LIN {X 0,Y 566.195,Z 141.956,A -85,B 0,C 180,E1 -2380.2,E2 -2380.2} C_VEL
LIN {X 0,Y 566.194,Z 141.961,A -85,B 0,C 180,E1 -2383.055,E2 -2383.055} C_VEL
LIN {X 0,Y 566.193,Z 141.957,A -85,B 0,C 180,E1 -2386.049,E2 -2386.049} C_VEL
LIN {X 0,Y 566.204,Z 141.954,A -85,B 0,C 180,E1 -2388.865,E2 -2388.865} C_VEL
LIN {X 0,Y 566.171,Z 141.963,A -85,B 0,C 180,E1 -2391.638,E2 -2391.638} C_VEL
LIN {X 0,Y 566.142,Z 141.962,A -85,B 0,C 180,E1 -2394.308,E2 -2394.308} C_VEL
LIN {X 0,Y 566.223,Z 141.954,A -85,B 0,C 180,E1 -2396.9,E2 -2396.9} C_VEL
LIN {X 0,Y 566.19,Z 141.957,A -85,B 0,C 180,E1 -2399.41,E2 -2399.41} C_VEL
LIN {X 0,Y 566.224,Z 141.955,A -85,B 0,C 180,E1 -2401.86,E2 -2401.86} C_VEL
LIN {X 0,Y 566.194,Z 141.955,A -85,B 0,C 180,E1 -2404.252,E2 -2404.252} C_VEL
LIN {X 0,Y 566.159,Z 141.959,A -85,B 0,C 180,E1 -2407.369,E2 -2407.369} C_VEL
LIN {X 0,Y 566.209,Z 141.956,A -85,B 0,C 180,E1 -2409.664,E2 -2409.664} C_VEL
LIN {X 0,Y 566.199,Z 141.955,A -85,B 0,C 180,E1 -2412.67,E2 -2412.67} C_VEL
LIN {X 0,Y 566.213,Z 141.953,A -85,B 0,C 180,E1 -2415.628,E2 -2415.628} C_VEL
LIN {X 0,Y 566.234,Z 141.952,A -85,B 0,C 180,E1 -2418.677,E2 -2418.677} C_VEL
LIN {X 0,Y 566.224,Z 141.954,A -85,B 0,C 180,E1 -2421.435,E2 -2421.435} C_VEL
LIN {X 0,Y 566.261,Z 141.947,A -85,B 0,C 180,E1 -2424.303,E2 -2424.303} C_VEL
LIN {X 0,Y 566.283,Z 141.945,A -85,B 0,C 180,E1 -2427.867,E2 -2427.867} C_VEL
LIN {X 0,Y 566.288,Z 141.949,A -85,B 0,C 180,E1 -2430.001,E2 -2430.001} C_VEL
LIN {X 0,Y 566.258,Z 141.947,A -85,B 0,C 180,E1 -2432.847,E2 -2432.847} C_VEL
LIN {X 0,Y 566.263,Z 141.948,A -85,B 0,C 180,E1 -2435.699,E2 -2435.699} C_VEL
LIN {X 0,Y 566.23,Z 141.956,A -85,B 0,C 180,E1 -2438.567,E2 -2438.567} C_VEL
LIN {X 0,Y 566.243,Z 141.951,A -85,B 0,C 180,E1 -2441.455,E2 -2441.455} C_VEL
LIN {X 0,Y 566.206,Z 141.953,A -85,B 0,C 180,E1 -2444.494,E2 -2444.494} C_VEL
LIN {X 0,Y 566.203,Z 141.956,A -85,B 0,C 180,E1 -2447.332,E2 -2447.332} C_VEL
LIN {X 0,Y 566.212,Z 141.959,A -85,B 0,C 180,E1 -2450.338,E2 -2450.338} C_VEL
LIN {X 0,Y 566.169,Z 141.961,A -85,B 0,C 180,E1 -2453.28,E2 -2453.28} C_VEL
LIN {X 0,Y 566.186,Z 141.957,A -85,B 0,C 180,E1 -2455.751,E2 -2455.751} C_VEL
LIN {X 0,Y 566.157,Z 141.961,A -85,B 0,C 180,E1 -2458.193,E2 -2458.193} C_VEL
LIN {X 0,Y 566.192,Z 141.955,A -85,B 0,C 180,E1 -2461.076,E2 -2461.076} C_VEL
LIN {X 0,Y 566.202,Z 141.96,A -85,B 0,C 180,E1 -2463.732,E2 -2463.732} C_VEL
LIN {X 0,Y 566.183,Z 141.958,A -85,B 0,C 180,E1 -2466.572,E2 -2466.572} C_VEL
LIN {X 0,Y 566.21,Z 141.953,A -85,B 0,C 180,E1 -2469.685,E2 -2469.685} C_VEL
LIN {X 0,Y 566.205,Z 141.954,A -85,B 0,C 180,E1 -2473.055,E2 -2473.055} C_VEL
LIN {X 0,Y 566.198,Z 141.955,A -85,B 0,C 180,E1 -2476.05,E2 -2476.05} C_VEL
LIN {X 0,Y 566.208,Z 141.955,A -85,B 0,C 180,E1 -2479.215,E2 -2479.215} C_VEL
LIN {X 0,Y 566.173,Z 141.958,A -85,B 0,C 180,E1 -2481.636,E2 -2481.636} C_VEL
LIN {X 0,Y 566.153,Z 141.961,A -85,B 0,C 180,E1 -2484.307,E2 -2484.307} C_VEL
LIN {X 0,Y 566.204,Z 141.957,A -85,B 0,C 180,E1 -2486.897,E2 -2486.897} C_VEL
LIN {X 0,Y 566.232,Z 142.057,A -85,B 0,C 180,E1 -2489.617,E2 -2489.617} C_VEL
LIN {X 0,Y 566.413,Z 147.475,A -85,B 0,C 180,E1 -2491.453,E2 -2491.453} C_VEL
LIN {X 0,Y 566.3,Z 155.916,A -85,B 0,C 180,E1 -2494.255,E2 -2494.255} C_VEL
LIN {X 0,Y 566.217,Z 164.488,A -85,B 0,C 180,E1 -2497.043,E2 -2497.043} C_VEL
LIN {X 0,Y 566.168,Z 173.964,A -85,B 0,C 180,E1 -2500.04,E2 -2500.04} C_VEL
LIN {X 0,Y 566.089,Z 183.007,A -85,B 0,C 180,E1 -2502.933,E2 -2502.933} C_VEL
LIN {X 0,Y 566.022,Z 192.721,A -85,B 0,C 180,E1 -2505.988,E2 -2505.988} C_VEL
LIN {X 0,Y 565.964,Z 201.9,A -85,B 0,C 180,E1 -2508.816,E2 -2508.816} C_VEL
LIN {X 0,Y 565.944,Z 211.648,A -85,B 0,C 180,E1 -2511.79,E2 -2511.79} C_VEL
LIN {X 0,Y 565.895,Z 214.384,A -85,B 0,C 180,E1 -2512.619,E2 -2512.619} C_VEL
LIN {X 0,Y 566.251,Z 220.58,A -85,B 0,C 180,E1 -2512.826,E2 -2512.826} C_VEL
LIN {X 0,Y 566.159,Z 229.406,A -85,B 0,C 180,E1 -2513.205,E2 -2513.205} C_VEL
LIN {X 0,Y 566.081,Z 238.598,A -85,B 0,C 180,E1 -2513.764,E2 -2513.764} C_VEL
LIN {X 0,Y 565.989,Z 245.323,A -85,B 0,C 180,E1 -2514.299,E2 -2514.299} C_VEL
LIN {X 0,Y 566.009,Z 252.383,A -85,B 0,C 180,E1 -2515.014,E2 -2515.014} C_VEL
LIN {X 0,Y 565.97,Z 257.771,A -85,B 0,C 180,E1 -2515.727,E2 -2515.727} C_VEL
LIN {X 0,Y 565.969,Z 262.032,A -85,B 0,C 180,E1 -2516.44,E2 -2516.44} C_VEL
LIN {X 0,Y 565.892,Z 265.349,A -85,B 0,C 180,E1 -2517.153,E2 -2517.153} C_VEL
LIN {X 0,Y 565.855,Z 267.84,A -85,B 0,C 180,E1 -2517.865,E2 -2517.865} C_VEL
LIN {X 0,Y 565.847,Z 269.58,A -85,B 0,C 180,E1 -2518.577,E2 -2518.577} C_VEL
LIN {X 0,Y 565.842,Z 270.622,A -85,B 0,C 180,E1 -2519.288,E2 -2519.288} C_VEL
LIN {X 0,Y 565.839,Z 270.996,A -85,B 0,C 180,E1 -2520,E2 -2520} C_VEL
LIN {X 0,Y 565.841,Z 270.711,A -85,B 0,C 180,E1 -2520.712,E2 -2520.712} C_VEL
LIN {X 0,Y 565.848,Z 269.761,A -85,B 0,C 180,E1 -2521.423,E2 -2521.423} C_VEL
LIN {X 0,Y 565.854,Z 268.12,A -85,B 0,C 180,E1 -2522.135,E2 -2522.135} C_VEL
LIN {X 0,Y 565.893,Z 265.732,A -85,B 0,C 180,E1 -2522.848,E2 -2522.848} C_VEL
LIN {X 0,Y 565.991,Z 260.601,A -85,B 0,C 180,E1 -2523.916,E2 -2523.916} C_VEL
LIN {X 0,Y 566.024,Z 254.526,A -85,B 0,C 180,E1 -2524.808,E2 -2524.808} C_VEL
LIN {X 0,Y 565.96,Z 248.211,A -85,B 0,C 180,E1 -2525.523,E2 -2525.523} C_VEL
LIN {X 0,Y 566.069,Z 241.059,A -85,B 0,C 180,E1 -2526.147,E2 -2526.147} C_VEL
LIN {X 0,Y 566.09,Z 233.058,A -85,B 0,C 180,E1 -2526.683,E2 -2526.683} C_VEL
LIN {X 0,Y 566.211,Z 224.178,A -85,B 0,C 180,E1 -2527.13,E2 -2527.13} C_VEL
LIN {X 0,Y 566.062,Z 216.549,A -85,B 0,C 180,E1 -2527.401,E2 -2527.401} C_VEL
LIN {X 0,Y 565.899,Z 214.311,A -85,B 0,C 180,E1 -2527.493,E2 -2527.493} C_VEL
LIN {X 0,Y 565.944,Z 204.843,A -85,B 0,C 180,E1 -2530.374,E2 -2530.374} C_VEL
LIN {X 0,Y 566.004,Z 195.375,A -85,B 0,C 180,E1 -2533.28,E2 -2533.28} C_VEL
LIN {X 0,Y 566.052,Z 187.164,A -85,B 0,C 180,E1 -2535.852,E2 -2535.852} C_VEL
LIN {X 0,Y 566.16,Z 177.828,A -85,B 0,C 180,E1 -2538.829,E2 -2538.829} C_VEL
LIN {X 0,Y 566.197,Z 168.251,A -85,B 0,C 180,E1 -2541.863,E2 -2541.863} C_VEL
LIN {X 0,Y 566.261,Z 158.561,A -85,B 0,C 180,E1 -2544.96,E2 -2544.96} C_VEL
LIN {X 0,Y 566.335,Z 149.951,A -85,B 0,C 180,E1 -2547.734,E2 -2547.734} C_VEL
LIN {X 0,Y 566.402,Z 143.716,A -85,B 0,C 180,E1 -2549.757,E2 -2549.757} C_VEL
LIN {X 0,Y 566.261,Z 141.954,A -85,B 0,C 180,E1 -2550.382,E2 -2550.382} C_VEL
LIN {X 0,Y 566.208,Z 141.958,A -85,B 0,C 180,E1 -2553.103,E2 -2553.103} C_VEL
LIN {X 0,Y 566.168,Z 141.964,A -85,B 0,C 180,E1 -2555.692,E2 -2555.692} C_VEL
LIN {X 0,Y 566.215,Z 141.957,A -85,B 0,C 180,E1 -2558.558,E2 -2558.558} C_VEL
LIN {X 0,Y 566.178,Z 141.962,A -85,B 0,C 180,E1 -2561.14,E2 -2561.14} C_VEL
LIN {X 0,Y 566.198,Z 141.959,A -85,B 0,C 180,E1 -2564.036,E2 -2564.036} C_VEL
LIN {X 0,Y 566.208,Z 141.959,A -85,B 0,C 180,E1 -2567.082,E2 -2567.082} C_VEL
LIN {X 0,Y 566.219,Z 141.958,A -85,B 0,C 180,E1 -2570.314,E2 -2570.314} C_VEL
LIN {X 0,Y 566.205,Z 141.96,A -85,B 0,C 180,E1 -2573.43,E2 -2573.43} C_VEL
LIN {X 0,Y 566.204,Z 141.959,A -85,B 0,C 180,E1 -2576.268,E2 -2576.268} C_VEL
LIN {X 0,Y 566.197,Z 141.963,A -85,B 0,C 180,E1 -2578.923,E2 -2578.923} C_VEL
LIN {X 0,Y 566.218,Z 141.96,A -85,B 0,C 180,E1 -2581.857,E2 -2581.857} C_VEL
LIN {X 0,Y 566.268,Z 142.067,A -85,B 0,C 180,E1 -2582.262,E2 -2582.262} C_VEL
LIN {X 0,Y 567.185,Z 147.623,A -85,B 0,C 180,E1 -2583.507,E2 -2583.507} C_VEL
LIN {X 0,Y 566.963,Z 159.309,A -85,B 0,C 180,E1 -2585.853,E2 -2585.853} C_VEL
LIN {X 0,Y 566.676,Z 173.884,A -85,B 0,C 180,E1 -2588.687,E2 -2588.687} C_VEL
LIN {X 0,Y 566.475,Z 189.392,A -85,B 0,C 180,E1 -2591.556,E2 -2591.556} C_VEL
LIN {X 0,Y 566.325,Z 204.592,A -85,B 0,C 180,E1 -2594.34,E2 -2594.34} C_VEL
LIN {X 0,Y 566.205,Z 219.792,A -85,B 0,C 180,E1 -2597.089,E2 -2597.089} C_VEL
LIN {X 0,Y 566.177,Z 221.014,A -85,B 0,C 180,E1 -2597.293,E2 -2597.293} C_VEL
LIN {X 0,Y 566.981,Z 226.896,A -85,B 0,C 180,E1 -2597.403,E2 -2597.403} C_VEL
LIN {X 0,Y 566.85,Z 239.423,A -85,B 0,C 180,E1 -2597.695,E2 -2597.695} C_VEL
LIN {X 0,Y 566.733,Z 252.352,A -85,B 0,C 180,E1 -2598.147,E2 -2598.147} C_VEL
LIN {X 0,Y 566.594,Z 264.395,A -85,B 0,C 180,E1 -2598.721,E2 -2598.721} C_VEL
LIN {X 0,Y 566.457,Z 276.184,A -85,B 0,C 180,E1 -2599.454,E2 -2599.454} C_VEL
LIN {X 0,Y 566.327,Z 286.591,A -85,B 0,C 180,E1 -2600.264,E2 -2600.264} C_VEL
LIN {X 0,Y 566.207,Z 295.103,A -85,B 0,C 180,E1 -2601.073,E2 -2601.073} C_VEL
LIN {X 0,Y 566.113,Z 302.952,A -85,B 0,C 180,E1 -2601.971,E2 -2601.971} C_VEL
LIN {X 0,Y 566.005,Z 310.616,A -85,B 0,C 180,E1 -2603.046,E2 -2603.046} C_VEL
LIN {X 0,Y 566.004,Z 317.674,A -85,B 0,C 180,E1 -2604.298,E2 -2604.298} C_VEL
LIN {X 0,Y 565.933,Z 322.368,A -85,B 0,C 180,E1 -2605.369,E2 -2605.369} C_VEL
LIN {X 0,Y 565.927,Z 325.955,A -85,B 0,C 180,E1 -2606.439,E2 -2606.439} C_VEL
LIN {X 0,Y 565.878,Z 327.805,A -85,B 0,C 180,E1 -2607.151,E2 -2607.151} C_VEL
LIN {X 0,Y 565.846,Z 330.183,A -85,B 0,C 180,E1 -2608.575,E2 -2608.575} C_VEL
LIN {X 0,Y 565.839,Z 331,A -85,B 0,C 180,E1 -2609.999,E2 -2609.999} C_VEL
LIN {X 0,Y 565.846,Z 330.187,A -85,B 0,C 180,E1 -2611.422,E2 -2611.422} C_VEL
LIN {X 0,Y 565.877,Z 327.813,A -85,B 0,C 180,E1 -2612.846,E2 -2612.846} C_VEL
LIN {X 0,Y 565.926,Z 324.9,A -85,B 0,C 180,E1 -2613.915,E2 -2613.915} C_VEL
LIN {X 0,Y 565.877,Z 320.954,A -85,B 0,C 180,E1 -2614.986,E2 -2614.986} C_VEL
LIN {X 0,Y 566.007,Z 315.874,A -85,B 0,C 180,E1 -2616.057,E2 -2616.057} C_VEL
LIN {X 0,Y 566.039,Z 309.476,A -85,B 0,C 180,E1 -2617.131,E2 -2617.131} C_VEL
LIN {X 0,Y 566.133,Z 301.488,A -85,B 0,C 180,E1 -2618.206,E2 -2618.206} C_VEL
LIN {X 0,Y 566.228,Z 293.347,A -85,B 0,C 180,E1 -2619.104,E2 -2619.104} C_VEL
LIN {X 0,Y 566.34,Z 283.415,A -85,B 0,C 180,E1 -2620.004,E2 -2620.004} C_VEL
LIN {X 0,Y 566.519,Z 272.33,A -85,B 0,C 180,E1 -2620.805,E2 -2620.805} C_VEL
LIN {X 0,Y 566.61,Z 261.199,A -85,B 0,C 180,E1 -2621.445,E2 -2621.445} C_VEL
LIN {X 0,Y 566.738,Z 249.013,A -85,B 0,C 180,E1 -2621.987,E2 -2621.987} C_VEL
LIN {X 0,Y 566.857,Z 236.227,A -85,B 0,C 180,E1 -2622.393,E2 -2622.393} C_VEL
LIN {X 0,Y 566.84,Z 225.151,A -85,B 0,C 180,E1 -2622.629,E2 -2622.629} C_VEL
LIN {X 0,Y 566.184,Z 220.818,A -85,B 0,C 180,E1 -2622.727,E2 -2622.727} C_VEL
LIN {X 0,Y 566.298,Z 205.618,A -85,B 0,C 180,E1 -2625.474,E2 -2625.474} C_VEL
LIN {X 0,Y 566.449,Z 190.418,A -85,B 0,C 180,E1 -2628.256,E2 -2628.256} C_VEL
LIN {X 0,Y 566.615,Z 177.294,A -85,B 0,C 180,E1 -2630.7,E2 -2630.7} C_VEL
LIN {X 0,Y 566.822,Z 164.181,A -85,B 0,C 180,E1 -2633.181,E2 -2633.181} C_VEL
LIN {X 0,Y 567.057,Z 150.067,A -85,B 0,C 180,E1 -2635.904,E2 -2635.904} C_VEL
LIN {X 0,Y 566.769,Z 144.561,A -85,B 0,C 180,E1 -2637.002,E2 -2637.002} C_VEL
LIN {X 0,Y 566.238,Z 141.954,A -85,B 0,C 180,E1 -2637.587,E2 -2637.587} C_VEL
LIN {X 0,Y 566.163,Z 141.965,A -85,B 0,C 180,E1 -2640.592,E2 -2640.592} C_VEL
LIN {X 0,Y 566.223,Z 141.952,A -85,B 0,C 180,E1 -2643.1,E2 -2643.1} C_VEL
LIN {X 0,Y 566.208,Z 141.96,A -85,B 0,C 180,E1 -2645.687,E2 -2645.687} C_VEL
LIN {X 0,Y 566.204,Z 141.955,A -85,B 0,C 180,E1 -2648.557,E2 -2648.557} C_VEL
LIN {X 0,Y 566.157,Z 141.962,A -85,B 0,C 180,E1 -2651.139,E2 -2651.139} C_VEL
LIN {X 0,Y 566.184,Z 141.961,A -85,B 0,C 180,E1 -2654.035,E2 -2654.035} C_VEL
LIN {X 0,Y 566.196,Z 141.957,A -85,B 0,C 180,E1 -2657.081,E2 -2657.081} C_VEL
LIN {X 0,Y 566.217,Z 141.953,A -85,B 0,C 180,E1 -2659.802,E2 -2659.802} C_VEL
LIN {X 0,Y 566.181,Z 141.963,A -85,B 0,C 180,E1 -2662.599,E2 -2662.599} C_VEL
LIN {X 0,Y 566.195,Z 141.96,A -85,B 0,C 180,E1 -2666.043,E2 -2666.043} C_VEL
LIN {X 0,Y 566.193,Z 141.955,A -85,B 0,C 180,E1 -2668.578,E2 -2668.578} C_VEL
LIN {X 0,Y 566.186,Z 141.962,A -85,B 0,C 180,E1 -2671.046,E2 -2671.046} C_VEL
LIN {X 0,Y 566.235,Z 141.95,A -85,B 0,C 180,E1 -2673.46,E2 -2673.46} C_VEL
LIN {X 0,Y 566.183,Z 141.961,A -85,B 0,C 180,E1 -2675.818,E2 -2675.818} C_VEL
LIN {X 0,Y 566.194,Z 141.956,A -85,B 0,C 180,E1 -2678.902,E2 -2678.902} C_VEL
LIN {X 0,Y 566.201,Z 141.959,A -85,B 0,C 180,E1 -2681.172,E2 -2681.172} C_VEL
LIN {X 0,Y 566.211,Z 141.953,A -85,B 0,C 180,E1 -2683.412,E2 -2683.412} C_VEL
LIN {X 0,Y 566.191,Z 141.958,A -85,B 0,C 180,E1 -2686.359,E2 -2686.359} C_VEL
LIN {X 0,Y 566.218,Z 141.952,A -85,B 0,C 180,E1 -2688.675,E2 -2688.675} C_VEL
LIN {X 0,Y 566.205,Z 141.956,A -85,B 0,C 180,E1 -2691.434,E2 -2691.434} C_VEL
LIN {X 0,Y 566.249,Z 141.953,A -85,B 0,C 180,E1 -2694.302,E2 -2694.302} C_VEL
LIN {X 0,Y 566.27,Z 141.951,A -85,B 0,C 180,E1 -2697.866,E2 -2697.866} C_VEL
LIN {X 0,Y 566.286,Z 141.945,A -85,B 0,C 180,E1 -2700.711,E2 -2700.711} C_VEL
LIN {X 0,Y 566.16,Z 141.959,A -85,B 0,C 180,E1 -2703.558,E2 -2703.558} C_VEL
LIN {X 0,Y 566.243,Z 141.95,A -85,B 0,C 180,E1 -2705.698,E2 -2705.698} C_VEL
LIN {X 0,Y 566.239,Z 141.95,A -85,B 0,C 180,E1 -2708.566,E2 -2708.566} C_VEL
LIN {X 0,Y 566.236,Z 141.954,A -85,B 0,C 180,E1 -2711.454,E2 -2711.454} C_VEL
LIN {X 0,Y 566.213,Z 141.958,A -85,B 0,C 180,E1 -2714.505,E2 -2714.505} C_VEL
LIN {X 0,Y 566.19,Z 141.956,A -85,B 0,C 180,E1 -2717.332,E2 -2717.332} C_VEL
LIN {X 0,Y 566.207,Z 141.954,A -85,B 0,C 180,E1 -2720.337,E2 -2720.337} C_VEL
LIN {X 0,Y 566.217,Z 141.954,A -85,B 0,C 180,E1 -2723.403,E2 -2723.403} C_VEL
LIN {X 0,Y 566.192,Z 141.956,A -85,B 0,C 180,E1 -2725.75,E2 -2725.75} C_VEL
LIN {X 0,Y 566.149,Z 141.96,A -85,B 0,C 180,E1 -2727.502,E2 -2727.502} C_VEL
LIN {X 0,Y 565.482,Z 142.049,A -85,B 0,C 180,E1 -2728.096,E2 -2728.096} C_VEL
LIN {X 0,Y 562.634,Z 142.399,A -85,B 0,C 180,E1 -2729.06,E2 -2729.06} C_VEL
LIN {X 0,Y 560.235,Z 142.702,A -85,B 0,C 180,E1 -2729.836,E2 -2729.836} C_VEL
LIN {X 0,Y 559.214,Z 142.825,A -85,B 0,C 180,E1 -2730.435,E2 -2730.435} C_VEL
LIN {X 0,Y 559.136,Z 142.834,A -85,B 0,C 180,E1 -2730.638,E2 -2730.638} C_VEL
LIN {X 0,Y 559.166,Z 142.832,A -85,B 0,C 180,E1 -2733.575,E2 -2733.575} C_VEL
LIN {X 0,Y 559.158,Z 142.837,A -85,B 0,C 180,E1 -2736.45,E2 -2736.45} C_VEL
LIN {X 0,Y 559.161,Z 142.831,A -85,B 0,C 180,E1 -2738.935,E2 -2738.935} C_VEL
LIN {X 0,Y 559.151,Z 142.835,A -85,B 0,C 180,E1 -2741.771,E2 -2741.771} C_VEL
LIN {X 0,Y 559.145,Z 142.834,A -85,B 0,C 180,E1 -2744.241,E2 -2744.241} C_VEL
LIN {X 0,Y 559.155,Z 142.832,A -85,B 0,C 180,E1 -2747.258,E2 -2747.258} C_VEL
LIN {X 0,Y 559.171,Z 142.833,A -85,B 0,C 180,E1 -2750.136,E2 -2750.136} C_VEL
LIN {X 0,Y 559.122,Z 142.839,A -85,B 0,C 180,E1 -2752.892,E2 -2752.892} C_VEL
LIN {X 0,Y 559.16,Z 142.832,A -85,B 0,C 180,E1 -2756.052,E2 -2756.052} C_VEL
LIN {X 0,Y 559.162,Z 142.831,A -85,B 0,C 180,E1 -2758.983,E2 -2758.983} C_VEL
LIN {X 0,Y 559.164,Z 142.836,A -85,B 0,C 180,E1 -2761.62,E2 -2761.62} C_VEL
LIN {X 0,Y 559.167,Z 142.83,A -85,B 0,C 180,E1 -2763.904,E2 -2763.904} C_VEL
LIN {X 0,Y 559.107,Z 142.839,A -85,B 0,C 180,E1 -2767.068,E2 -2767.068} C_VEL
LIN {X 0,Y 559.176,Z 142.83,A -85,B 0,C 180,E1 -2769.397,E2 -2769.397} C_VEL
LIN {X 0,Y 559.146,Z 142.839,A -85,B 0,C 180,E1 -2771.687,E2 -2771.687} C_VEL
LIN {X 0,Y 559.163,Z 142.832,A -85,B 0,C 180,E1 -2773.949,E2 -2773.949} C_VEL
LIN {X 0,Y 559.149,Z 142.834,A -85,B 0,C 180,E1 -2776.185,E2 -2776.185} C_VEL
LIN {X 0,Y 559.19,Z 142.827,A -85,B 0,C 180,E1 -2779.135,E2 -2779.135} C_VEL
LIN {X 0,Y 559.2,Z 142.829,A -85,B 0,C 180,E1 -2782.055,E2 -2782.055} C_VEL
LIN {X 0,Y 559.252,Z 142.825,A -85,B 0,C 180,E1 -2784.955,E2 -2784.955} C_VEL
LIN {X 0,Y 559.254,Z 142.82,A -85,B 0,C 180,E1 -2787.841,E2 -2787.841} C_VEL
LIN {X 0,Y 559.256,Z 142.824,A -85,B 0,C 180,E1 -2790.001,E2 -2790.001} C_VEL
LIN {X 0,Y 559.226,Z 142.823,A -85,B 0,C 180,E1 -2792.883,E2 -2792.883} C_VEL
LIN {X 0,Y 559.232,Z 142.823,A -85,B 0,C 180,E1 -2795.771,E2 -2795.771} C_VEL
LIN {X 0,Y 559.188,Z 142.833,A -85,B 0,C 180,E1 -2798.675,E2 -2798.675} C_VEL
LIN {X 0,Y 559.2,Z 142.83,A -85,B 0,C 180,E1 -2801.602,E2 -2801.602} C_VEL
LIN {X 0,Y 559.156,Z 142.832,A -85,B 0,C 180,E1 -2804.577,E2 -2804.577} C_VEL
LIN {X 0,Y 559.146,Z 142.833,A -85,B 0,C 180,E1 -2807.558,E2 -2807.558} C_VEL
LIN {X 0,Y 559.171,Z 142.832,A -85,B 0,C 180,E1 -2809.838,E2 -2809.838} C_VEL
LIN {X 0,Y 559.137,Z 142.838,A -85,B 0,C 180,E1 -2812.154,E2 -2812.154} C_VEL
LIN {X 0,Y 559.142,Z 142.839,A -85,B 0,C 180,E1 -2815.178,E2 -2815.178} C_VEL
LIN {X 0,Y 559.119,Z 142.836,A -85,B 0,C 180,E1 -2817.716,E2 -2817.716} C_VEL
LIN {X 0,Y 559.143,Z 142.838,A -85,B 0,C 180,E1 -2820.184,E2 -2820.184} C_VEL
LIN {X 0,Y 559.157,Z 142.832,A -85,B 0,C 180,E1 -2822.716,E2 -2822.716} C_VEL
LIN {X 0,Y 559.128,Z 142.842,A -85,B 0,C 180,E1 -2825.325,E2 -2825.325} C_VEL
LIN {X 0,Y 559.11,Z 142.837,A -85,B 0,C 180,E1 -2828.02,E2 -2828.02} C_VEL
LIN {X 0,Y 559.159,Z 142.832,A -85,B 0,C 180,E1 -2829.941,E2 -2829.941} C_VEL
LIN {X 0,Y 559.161,Z 142.832,A -85,B 0,C 180,E1 -2832.744,E2 -2832.744} C_VEL
LIN {X 0,Y 559.152,Z 142.835,A -85,B 0,C 180,E1 -2835.762,E2 -2835.762} C_VEL
LIN {X 0,Y 559.166,Z 142.831,A -85,B 0,C 180,E1 -2838.23,E2 -2838.23} C_VEL
LIN {X 0,Y 559.169,Z 142.829,A -85,B 0,C 180,E1 -2841.193,E2 -2841.193} C_VEL
LIN {X 0,Y 559.123,Z 142.842,A -85,B 0,C 180,E1 -2843.788,E2 -2843.788} C_VEL
LIN {X 0,Y 559.151,Z 142.833,A -85,B 0,C 180,E1 -2846.424,E2 -2846.424} C_VEL
LIN {X 0,Y 559.213,Z 142.917,A -85,B 0,C 180,E1 -2849.508,E2 -2849.508} C_VEL
LIN {X 0,Y 559.399,Z 147.468,A -85,B 0,C 180,E1 -2851.073,E2 -2851.073} C_VEL
LIN {X 0,Y 559.291,Z 155.893,A -85,B 0,C 180,E1 -2853.908,E2 -2853.908} C_VEL
LIN {X 0,Y 559.165,Z 163.968,A -85,B 0,C 180,E1 -2856.567,E2 -2856.567} C_VEL
LIN {X 0,Y 559.132,Z 172.758,A -85,B 0,C 180,E1 -2859.394,E2 -2859.394} C_VEL
LIN {X 0,Y 559.041,Z 181.068,A -85,B 0,C 180,E1 -2862.061,E2 -2862.061} C_VEL
LIN {X 0,Y 558.988,Z 189.275,A -85,B 0,C 180,E1 -2864.691,E2 -2864.691} C_VEL
LIN {X 0,Y 558.935,Z 197.495,A -85,B 0,C 180,E1 -2867.288,E2 -2867.288} C_VEL
LIN {X 0,Y 558.864,Z 206.917,A -85,B 0,C 180,E1 -2870.226,E2 -2870.226} C_VEL
LIN {X 0,Y 558.832,Z 214.386,A -85,B 0,C 180,E1 -2872.526,E2 -2872.526} C_VEL
LIN {X 0,Y 559.208,Z 221.803,A -85,B 0,C 180,E1 -2872.78,E2 -2872.78} C_VEL
LIN {X 0,Y 559.111,Z 230.589,A -85,B 0,C 180,E1 -2873.178,E2 -2873.178} C_VEL
LIN {X 0,Y 559.039,Z 238.604,A -85,B 0,C 180,E1 -2873.685,E2 -2873.685} C_VEL
LIN {X 0,Y 558.935,Z 245.327,A -85,B 0,C 180,E1 -2874.227,E2 -2874.227} C_VEL
LIN {X 0,Y 558.929,Z 252.388,A -85,B 0,C 180,E1 -2874.95,E2 -2874.95} C_VEL
LIN {X 0,Y 558.907,Z 257.774,A -85,B 0,C 180,E1 -2875.673,E2 -2875.673} C_VEL
LIN {X 0,Y 558.882,Z 262.035,A -85,B 0,C 180,E1 -2876.395,E2 -2876.395} C_VEL
LIN {X 0,Y 558.816,Z 265.352,A -85,B 0,C 180,E1 -2877.116,E2 -2877.116} C_VEL
LIN {X 0,Y 558.763,Z 267.843,A -85,B 0,C 180,E1 -2877.838,E2 -2877.838} C_VEL
LIN {X 0,Y 558.747,Z 269.582,A -85,B 0,C 180,E1 -2878.559,E2 -2878.559} C_VEL
LIN {X 0,Y 558.742,Z 270.623,A -85,B 0,C 180,E1 -2879.279,E2 -2879.279} C_VEL
LIN {X 0,Y 558.74,Z 270.996,A -85,B 0,C 180,E1 -2880,E2 -2880} C_VEL
LIN {X 0,Y 558.741,Z 270.71,A -85,B 0,C 180,E1 -2880.721,E2 -2880.721} C_VEL
LIN {X 0,Y 558.748,Z 269.759,A -85,B 0,C 180,E1 -2881.442,E2 -2881.442} C_VEL
LIN {X 0,Y 558.763,Z 268.118,A -85,B 0,C 180,E1 -2882.163,E2 -2882.163} C_VEL
LIN {X 0,Y 558.816,Z 265.73,A -85,B 0,C 180,E1 -2882.884,E2 -2882.884} C_VEL
LIN {X 0,Y 558.89,Z 260.598,A -85,B 0,C 180,E1 -2883.966,E2 -2883.966} C_VEL
LIN {X 0,Y 558.952,Z 254.521,A -85,B 0,C 180,E1 -2884.869,E2 -2884.869} C_VEL
LIN {X 0,Y 558.896,Z 248.204,A -85,B 0,C 180,E1 -2885.593,E2 -2885.593} C_VEL
LIN {X 0,Y 559.025,Z 241.053,A -85,B 0,C 180,E1 -2886.225,E2 -2886.225} C_VEL
LIN {X 0,Y 559.037,Z 232.936,A -85,B 0,C 180,E1 -2886.775,E2 -2886.775} C_VEL
LIN {X 0,Y 559.176,Z 224.165,A -85,B 0,C 180,E1 -2887.22,E2 -2887.22} C_VEL
LIN {X 0,Y 558.931,Z 215.697,A -85,B 0,C 180,E1 -2887.519,E2 -2887.519} C_VEL
LIN {X 0,Y 558.803,Z 214.309,A -85,B 0,C 180,E1 -2887.589,E2 -2887.589} C_VEL
LIN {X 0,Y 558.863,Z 204.841,A -85,B 0,C 180,E1 -2890.506,E2 -2890.506} C_VEL
LIN {X 0,Y 558.94,Z 195.462,A -85,B 0,C 180,E1 -2893.451,E2 -2893.451} C_VEL
LIN {X 0,Y 559.03,Z 186.106,A -85,B 0,C 180,E1 -2896.431,E2 -2896.431} C_VEL
LIN {X 0,Y 559.108,Z 177.94,A -85,B 0,C 180,E1 -2899.076,E2 -2899.076} C_VEL
LIN {X 0,Y 559.145,Z 170.146,A -85,B 0,C 180,E1 -2901.545,E2 -2901.545} C_VEL
LIN {X 0,Y 559.247,Z 160.994,A -85,B 0,C 180,E1 -2904.501,E2 -2904.501} C_VEL
LIN {X 0,Y 559.327,Z 152.415,A -85,B 0,C 180,E1 -2907.299,E2 -2907.299} C_VEL
LIN {X 0,Y 559.389,Z 144.546,A -85,B 0,C 180,E1 -2909.899,E2 -2909.899} C_VEL
LIN {X 0,Y 559.191,Z 142.834,A -85,B 0,C 180,E1 -2910.494,E2 -2910.494} C_VEL
LIN {X 0,Y 559.153,Z 142.838,A -85,B 0,C 180,E1 -2913.576,E2 -2913.576} C_VEL
LIN {X 0,Y 559.152,Z 142.837,A -85,B 0,C 180,E1 -2916.445,E2 -2916.445} C_VEL
LIN {X 0,Y 559.179,Z 142.834,A -85,B 0,C 180,E1 -2918.934,E2 -2918.934} C_VEL
LIN {X 0,Y 559.168,Z 142.835,A -85,B 0,C 180,E1 -2921.77,E2 -2921.77} C_VEL
LIN {X 0,Y 559.141,Z 142.84,A -85,B 0,C 180,E1 -2924.739,E2 -2924.739} C_VEL
LIN {X 0,Y 559.164,Z 142.835,A -85,B 0,C 180,E1 -2927.256,E2 -2927.256} C_VEL
LIN {X 0,Y 559.184,Z 142.835,A -85,B 0,C 180,E1 -2930.134,E2 -2930.134} C_VEL
LIN {X 0,Y 559.146,Z 142.837,A -85,B 0,C 180,E1 -2932.891,E2 -2932.891} C_VEL
LIN {X 0,Y 559.163,Z 142.836,A -85,B 0,C 180,E1 -2936.052,E2 -2936.052} C_VEL
LIN {X 0,Y 559.161,Z 142.84,A -85,B 0,C 180,E1 -2938.98,E2 -2938.98} C_VEL
LIN {X 0,Y 559.209,Z 142.911,A -85,B 0,C 180,E1 -2941.987,E2 -2941.987} C_VEL
LIN {X 0,Y 560.154,Z 147.894,A -85,B 0,C 180,E1 -2943.148,E2 -2943.148} C_VEL
LIN {X 0,Y 560.181,Z 154.731,A -85,B 0,C 180,E1 -2944.597,E2 -2944.597} C_VEL
LIN {X 0,Y 559.838,Z 167.218,A -85,B 0,C 180,E1 -2947.097,E2 -2947.097} C_VEL
LIN {X 0,Y 559.603,Z 182.102,A -85,B 0,C 180,E1 -2949.986,E2 -2949.986} C_VEL
LIN {X 0,Y 559.403,Z 196.824,A -85,B 0,C 180,E1 -2952.712,E2 -2952.712} C_VEL
LIN {X 0,Y 559.17,Z 212.202,A -85,B 0,C 180,E1 -2955.535,E2 -2955.535} C_VEL
LIN {X 0,Y 559.169,Z 221.014,A -85,B 0,C 180,E1 -2957.131,E2 -2957.131} C_VEL
LIN {X 0,Y 560.049,Z 228.038,A -85,B 0,C 180,E1 -2957.267,E2 -2957.267} C_VEL
LIN {X 0,Y 559.919,Z 240.946,A -85,B 0,C 180,E1 -2957.586,E2 -2957.586} C_VEL
LIN {X 0,Y 559.766,Z 253.473,A -85,B 0,C 180,E1 -2958.043,E2 -2958.043} C_VEL
LIN {X 0,Y 559.628,Z 265.407,A -85,B 0,C 180,E1 -2958.637,E2 -2958.637} C_VEL
LIN {X 0,Y 559.427,Z 277.472,A -85,B 0,C 180,E1 -2959.412,E2 -2959.412} C_VEL
LIN {X 0,Y 559.298,Z 287.635,A -85,B 0,C 180,E1 -2960.232,E2 -2960.232} C_VEL
LIN {X 0,Y 559.133,Z 296.777,A -85,B 0,C 180,E1 -2961.142,E2 -2961.142} C_VEL
LIN {X 0,Y 559.01,Z 305.681,A -85,B 0,C 180,E1 -2962.232,E2 -2962.232} C_VEL
LIN {X 0,Y 558.926,Z 311.733,A -85,B 0,C 180,E1 -2963.139,E2 -2963.139} C_VEL
LIN {X 0,Y 558.936,Z 317.674,A -85,B 0,C 180,E1 -2964.226,E2 -2964.226} C_VEL
LIN {X 0,Y 558.827,Z 322.368,A -85,B 0,C 180,E1 -2965.31,E2 -2965.31} C_VEL
LIN {X 0,Y 558.836,Z 325.955,A -85,B 0,C 180,E1 -2966.394,E2 -2966.394} C_VEL
LIN {X 0,Y 558.799,Z 327.805,A -85,B 0,C 180,E1 -2967.115,E2 -2967.115} C_VEL
LIN {X 0,Y 558.745,Z 330.182,A -85,B 0,C 180,E1 -2968.557,E2 -2968.557} C_VEL
LIN {X 0,Y 558.74,Z 331,A -85,B 0,C 180,E1 -2969.999,E2 -2969.999} C_VEL
LIN {X 0,Y 558.745,Z 330.186,A -85,B 0,C 180,E1 -2971.44,E2 -2971.44} C_VEL
LIN {X 0,Y 558.799,Z 327.813,A -85,B 0,C 180,E1 -2972.882,E2 -2972.882} C_VEL
LIN {X 0,Y 558.844,Z 324.899,A -85,B 0,C 180,E1 -2973.965,E2 -2973.965} C_VEL
LIN {X 0,Y 558.798,Z 320.954,A -85,B 0,C 180,E1 -2975.05,E2 -2975.05} C_VEL
LIN {X 0,Y 558.922,Z 315.874,A -85,B 0,C 180,E1 -2976.134,E2 -2976.134} C_VEL
LIN {X 0,Y 558.976,Z 309.475,A -85,B 0,C 180,E1 -2977.222,E2 -2977.222} C_VEL
LIN {X 0,Y 559.098,Z 301.488,A -85,B 0,C 180,E1 -2978.31,E2 -2978.31} C_VEL
LIN {X 0,Y 559.194,Z 293.346,A -85,B 0,C 180,E1 -2979.22,E2 -2979.22} C_VEL
LIN {X 0,Y 559.349,Z 283.414,A -85,B 0,C 180,E1 -2980.13,E2 -2980.13} C_VEL
LIN {X 0,Y 559.541,Z 272.427,A -85,B 0,C 180,E1 -2980.935,E2 -2980.935} C_VEL
LIN {X 0,Y 559.669,Z 260.484,A -85,B 0,C 180,E1 -2981.626,E2 -2981.626} C_VEL
LIN {X 0,Y 559.826,Z 247.804,A -85,B 0,C 180,E1 -2982.183,E2 -2982.183} C_VEL
LIN {X 0,Y 559.969,Z 234.397,A -85,B 0,C 180,E1 -2982.594,E2 -2982.594} C_VEL
LIN {X 0,Y 559.846,Z 225.694,A -85,B 0,C 180,E1 -2982.781,E2 -2982.781} C_VEL
LIN {X 0,Y 559.151,Z 220.818,A -85,B 0,C 180,E1 -2982.89,E2 -2982.89} C_VEL
LIN {X 0,Y 559.292,Z 205.618,A -85,B 0,C 180,E1 -2985.673,E2 -2985.673} C_VEL
LIN {X 0,Y 559.453,Z 190.304,A -85,B 0,C 180,E1 -2988.492,E2 -2988.492} C_VEL
LIN {X 0,Y 559.671,Z 177.281,A -85,B 0,C 180,E1 -2990.969,E2 -2990.969} C_VEL
LIN {X 0,Y 559.892,Z 165.414,A -85,B 0,C 180,E1 -2993.256,E2 -2993.256} C_VEL
LIN {X 0,Y 560.127,Z 153.074,A -85,B 0,C 180,E1 -2995.662,E2 -2995.662} C_VEL
LIN {X 0,Y 559.919,Z 146.518,A -85,B 0,C 180,E1 -2996.978,E2 -2996.978} C_VEL
LIN {X 0,Y 559.172,Z 142.835,A -85,B 0,C 180,E1 -2997.811,E2 -2997.811} C_VEL
LIN {X 0,Y 559.145,Z 142.837,A -85,B 0,C 180,E1 -3001.018,E2 -3001.018} C_VEL
LIN {X 0,Y 559.163,Z 142.836,A -85,B 0,C 180,E1 -3003.948,E2 -3003.948} C_VEL
LIN {X 0,Y 559.164,Z 142.831,A -85,B 0,C 180,E1 -3006.447,E2 -3006.447} C_VEL
LIN {X 0,Y 559.167,Z 142.835,A -85,B 0,C 180,E1 -3008.933,E2 -3008.933} C_VEL
LIN {X 0,Y 559.145,Z 142.833,A -85,B 0,C 180,E1 -3011.77,E2 -3011.77} C_VEL
LIN {X 0,Y 559.129,Z 142.836,A -85,B 0,C 180,E1 -3014.738,E2 -3014.738} C_VEL
LIN {X 0,Y 559.155,Z 142.836,A -85,B 0,C 180,E1 -3017.256,E2 -3017.256} C_VEL
LIN {X 0,Y 559.177,Z 142.829,A -85,B 0,C 180,E1 -3020.134,E2 -3020.134} C_VEL
LIN {X 0,Y 559.118,Z 142.839,A -85,B 0,C 180,E1 -3022.89,E2 -3022.89} C_VEL
LIN {X 0,Y 559.151,Z 142.837,A -85,B 0,C 180,E1 -3026.05,E2 -3026.05} C_VEL
LIN {X 0,Y 559.156,Z 142.835,A -85,B 0,C 180,E1 -3028.981,E2 -3028.981} C_VEL
LIN {X 0,Y 559.159,Z 142.832,A -85,B 0,C 180,E1 -3031.617,E2 -3031.617} C_VEL
LIN {X 0,Y 559.188,Z 142.83,A -85,B 0,C 180,E1 -3033.903,E2 -3033.903} C_VEL
LIN {X 0,Y 559.124,Z 142.836,A -85,B 0,C 180,E1 -3036.571,E2 -3036.571} C_VEL
LIN {X 0,Y 559.167,Z 142.837,A -85,B 0,C 180,E1 -3039.395,E2 -3039.395} C_VEL
LIN {X 0,Y 559.144,Z 142.834,A -85,B 0,C 180,E1 -3041.686,E2 -3041.686} C_VEL
LIN {X 0,Y 559.161,Z 142.833,A -85,B 0,C 180,E1 -3043.948,E2 -3043.948} C_VEL
LIN {X 0,Y 559.166,Z 142.836,A -85,B 0,C 180,E1 -3046.184,E2 -3046.184} C_VEL
LIN {X 0,Y 559.173,Z 142.833,A -85,B 0,C 180,E1 -3049.133,E2 -3049.133} C_VEL
LIN {X 0,Y 559.185,Z 142.828,A -85,B 0,C 180,E1 -3052.053,E2 -3052.053} C_VEL
LIN {X 0,Y 559.246,Z 142.822,A -85,B 0,C 180,E1 -3054.953,E2 -3054.953} C_VEL
LIN {X 0,Y 559.241,Z 142.827,A -85,B 0,C 180,E1 -3057.839,E2 -3057.839} C_VEL
LIN {X 0,Y 559.257,Z 142.821,A -85,B 0,C 180,E1 -3060.72,E2 -3060.72} C_VEL
LIN {X 0,Y 559.219,Z 142.83,A -85,B 0,C 180,E1 -3062.881,E2 -3062.881} C_VEL
LIN {X 0,Y 559.212,Z 142.826,A -85,B 0,C 180,E1 -3065.77,E2 -3065.77} C_VEL
LIN {X 0,Y 559.193,Z 142.827,A -85,B 0,C 180,E1 -3068.674,E2 -3068.674} C_VEL
LIN {X 0,Y 559.194,Z 142.829,A -85,B 0,C 180,E1 -3071.601,E2 -3071.601} C_VEL
LIN {X 0,Y 559.184,Z 142.835,A -85,B 0,C 180,E1 -3074.596,E2 -3074.596} C_VEL
LIN {X 0,Y 559.149,Z 142.835,A -85,B 0,C 180,E1 -3077.557,E2 -3077.557} C_VEL
LIN {X 0,Y 559.162,Z 142.835,A -85,B 0,C 180,E1 -3079.838,E2 -3079.838} C_VEL
LIN {X 0,Y 559.143,Z 142.834,A -85,B 0,C 180,E1 -3082.153,E2 -3082.153} C_VEL
LIN {X 0,Y 559.147,Z 142.838,A -85,B 0,C 180,E1 -3084.506,E2 -3084.506} C_VEL
LIN {X 0,Y 559.141,Z 142.834,A -85,B 0,C 180,E1 -3086.904,E2 -3086.904} C_VEL
LIN {X 0,Y 559.159,Z 142.836,A -85,B 0,C 180,E1 -3089.863,E2 -3089.863} C_VEL
LIN {X 0,Y 559.136,Z 142.834,A -85,B 0,C 180,E1 -3090.638,E2 -3090.638} C_VEL
LIN {X 0,Y 558.478,Z 142.922,A -85,B 0,C 180,E1 -3091.239,E2 -3091.239} C_VEL
LIN {X 0,Y 555.617,Z 143.275,A -85,B 0,C 180,E1 -3092.215,E2 -3092.215} C_VEL
LIN {X 0,Y 553.205,Z 143.579,A -85,B 0,C 180,E1 -3093.001,E2 -3093.001} C_VEL
LIN {X 0,Y 552.186,Z 143.701,A -85,B 0,C 180,E1 -3093.608,E2 -3093.608} C_VEL
LIN {X 0,Y 552.113,Z 143.71,A -85,B 0,C 180,E1 -3093.813,E2 -3093.813} C_VEL
LIN {X 0,Y 552.1,Z 143.713,A -85,B 0,C 180,E1 -3096.748,E2 -3096.748} C_VEL
LIN {X 0,Y 552.117,Z 143.712,A -85,B 0,C 180,E1 -3099.528,E2 -3099.528} C_VEL
LIN {X 0,Y 552.119,Z 143.708,A -85,B 0,C 180,E1 -3102.427,E2 -3102.427} C_VEL
LIN {X 0,Y 552.09,Z 143.712,A -85,B 0,C 180,E1 -3105.564,E2 -3105.564} C_VEL
LIN {X 0,Y 552.132,Z 143.708,A -85,B 0,C 180,E1 -3108.677,E2 -3108.677} C_VEL
LIN {X 0,Y 552.105,Z 143.716,A -85,B 0,C 180,E1 -3111.412,E2 -3111.412} C_VEL
LIN {X 0,Y 552.067,Z 143.715,A -85,B 0,C 180,E1 -3114.157,E2 -3114.157} C_VEL
LIN {X 0,Y 552.117,Z 143.712,A -85,B 0,C 180,E1 -3116.816,E2 -3116.816} C_VEL
LIN {X 0,Y 552.11,Z 143.711,A -85,B 0,C 180,E1 -3119.393,E2 -3119.393} C_VEL
LIN {X 0,Y 552.118,Z 143.711,A -85,B 0,C 180,E1 -3121.904,E2 -3121.904} C_VEL
LIN {X 0,Y 552.08,Z 143.716,A -85,B 0,C 180,E1 -3124.667,E2 -3124.667} C_VEL
LIN {X 0,Y 552.08,Z 143.713,A -85,B 0,C 180,E1 -3127.55,E2 -3127.55} C_VEL
LIN {X 0,Y 552.147,Z 143.707,A -85,B 0,C 180,E1 -3130.375,E2 -3130.375} C_VEL
LIN {X 0,Y 552.154,Z 143.707,A -85,B 0,C 180,E1 -3132.979,E2 -3132.979} C_VEL
LIN {X 0,Y 552.115,Z 143.709,A -85,B 0,C 180,E1 -3136.005,E2 -3136.005} C_VEL
LIN {X 0,Y 552.159,Z 143.703,A -85,B 0,C 180,E1 -3138.995,E2 -3138.995} C_VEL
LIN {X 0,Y 552.154,Z 143.708,A -85,B 0,C 180,E1 -3141.953,E2 -3141.953} C_VEL
LIN {X 0,Y 552.228,Z 143.7,A -85,B 0,C 180,E1 -3144.89,E2 -3144.89} C_VEL
LIN {X 0,Y 552.225,Z 143.696,A -85,B 0,C 180,E1 -3147.813,E2 -3147.813} C_VEL
LIN {X 0,Y 552.225,Z 143.7,A -85,B 0,C 180,E1 -3150.001,E2 -3150.001} C_VEL
LIN {X 0,Y 552.195,Z 143.7,A -85,B 0,C 180,E1 -3152.919,E2 -3152.919} C_VEL
LIN {X 0,Y 552.202,Z 143.699,A -85,B 0,C 180,E1 -3155.845,E2 -3155.845} C_VEL
LIN {X 0,Y 552.156,Z 143.707,A -85,B 0,C 180,E1 -3158.787,E2 -3158.787} C_VEL
LIN {X 0,Y 552.155,Z 143.709,A -85,B 0,C 180,E1 -3161.752,E2 -3161.752} C_VEL
LIN {X 0,Y 552.123,Z 143.709,A -85,B 0,C 180,E1 -3164.75,E2 -3164.75} C_VEL
LIN {X 0,Y 552.104,Z 143.71,A -85,B 0,C 180,E1 -3167.79,E2 -3167.79} C_VEL
LIN {X 0,Y 552.131,Z 143.712,A -85,B 0,C 180,E1 -3170.102,E2 -3170.102} C_VEL
LIN {X 0,Y 552.088,Z 143.713,A -85,B 0,C 180,E1 -3172.452,E2 -3172.452} C_VEL
LIN {X 0,Y 552.085,Z 143.718,A -85,B 0,C 180,E1 -3175.334,E2 -3175.334} C_VEL
LIN {X 0,Y 552.065,Z 143.716,A -85,B 0,C 180,E1 -3178.102,E2 -3178.102} C_VEL
LIN {X 0,Y 552.1,Z 143.714,A -85,B 0,C 180,E1 -3180.61,E2 -3180.61} C_VEL
LIN {X 0,Y 552.112,Z 143.711,A -85,B 0,C 180,E1 -3183.187,E2 -3183.187} C_VEL
LIN {X 0,Y 552.079,Z 143.715,A -85,B 0,C 180,E1 -3185.845,E2 -3185.845} C_VEL
LIN {X 0,Y 552.095,Z 143.713,A -85,B 0,C 180,E1 -3189.058,E2 -3189.058} C_VEL
LIN {X 0,Y 552.084,Z 143.713,A -85,B 0,C 180,E1 -3191.45,E2 -3191.45} C_VEL
LIN {X 0,Y 552.096,Z 143.712,A -85,B 0,C 180,E1 -3194.438,E2 -3194.438} C_VEL
LIN {X 0,Y 552.135,Z 143.708,A -85,B 0,C 180,E1 -3197.585,E2 -3197.585} C_VEL
LIN {X 0,Y 552.128,Z 143.714,A -85,B 0,C 180,E1 -3200.473,E2 -3200.473} C_VEL
LIN {X 0,Y 552.1,Z 143.712,A -85,B 0,C 180,E1 -3203.319,E2 -3203.319} C_VEL
LIN {X 0,Y 552.105,Z 143.712,A -85,B 0,C 180,E1 -3205.938,E2 -3205.938} C_VEL
LIN {X 0,Y 552.137,Z 143.712,A -85,B 0,C 180,E1 -3208.968,E2 -3208.968} C_VEL
LIN {X 0,Y 552.14,Z 143.775,A -85,B 0,C 180,E1 -3209.393,E2 -3209.393} C_VEL
LIN {X 0,Y 552.429,Z 147.429,A -85,B 0,C 180,E1 -3210.673,E2 -3210.673} C_VEL
LIN {X 0,Y 552.299,Z 155.87,A -85,B 0,C 180,E1 -3213.553,E2 -3213.553} C_VEL
LIN {X 0,Y 552.148,Z 164.463,A -85,B 0,C 180,E1 -3216.414,E2 -3216.414} C_VEL
LIN {X 0,Y 552.074,Z 173.968,A -85,B 0,C 180,E1 -3219.508,E2 -3219.508} C_VEL
LIN {X 0,Y 552,Z 182.316,A -85,B 0,C 180,E1 -3222.208,E2 -3222.208} C_VEL
LIN {X 0,Y 551.921,Z 191.698,A -85,B 0,C 180,E1 -3225.246,E2 -3225.246} C_VEL
LIN {X 0,Y 551.812,Z 201.097,A -85,B 0,C 180,E1 -3228.242,E2 -3228.242} C_VEL
LIN {X 0,Y 551.763,Z 209.334,A -85,B 0,C 180,E1 -3230.839,E2 -3230.839} C_VEL
LIN {X 0,Y 551.724,Z 214.45,A -85,B 0,C 180,E1 -3232.429,E2 -3232.429} C_VEL
LIN {X 0,Y 552.184,Z 222.009,A -85,B 0,C 180,E1 -3232.688,E2 -3232.688} C_VEL
LIN {X 0,Y 552.071,Z 230.712,A -85,B 0,C 180,E1 -3233.091,E2 -3233.091} C_VEL
LIN {X 0,Y 551.999,Z 238.732,A -85,B 0,C 180,E1 -3233.608,E2 -3233.608} C_VEL
LIN {X 0,Y 551.886,Z 245.374,A -85,B 0,C 180,E1 -3234.153,E2 -3234.153} C_VEL
LIN {X 0,Y 551.854,Z 252.402,A -85,B 0,C 180,E1 -3234.886,E2 -3234.886} C_VEL
LIN {X 0,Y 551.83,Z 257.777,A -85,B 0,C 180,E1 -3235.618,E2 -3235.618} C_VEL
LIN {X 0,Y 551.795,Z 262.037,A -85,B 0,C 180,E1 -3236.349,E2 -3236.349} C_VEL
LIN {X 0,Y 551.742,Z 265.355,A -85,B 0,C 180,E1 -3237.079,E2 -3237.079} C_VEL
LIN {X 0,Y 551.675,Z 267.845,A -85,B 0,C 180,E1 -3237.81,E2 -3237.81} C_VEL
LIN {X 0,Y 551.648,Z 269.584,A -85,B 0,C 180,E1 -3238.54,E2 -3238.54} C_VEL
LIN {X 0,Y 551.642,Z 270.624,A -85,B 0,C 180,E1 -3239.27,E2 -3239.27} C_VEL
LIN {X 0,Y 551.641,Z 270.996,A -85,B 0,C 180,E1 -3240,E2 -3240} C_VEL
LIN {X 0,Y 551.642,Z 270.709,A -85,B 0,C 180,E1 -3240.73,E2 -3240.73} C_VEL
LIN {X 0,Y 551.648,Z 269.758,A -85,B 0,C 180,E1 -3241.46,E2 -3241.46} C_VEL
LIN {X 0,Y 551.674,Z 268.117,A -85,B 0,C 180,E1 -3242.19,E2 -3242.19} C_VEL
LIN {X 0,Y 551.743,Z 265.728,A -85,B 0,C 180,E1 -3242.921,E2 -3242.921} C_VEL
LIN {X 0,Y 551.801,Z 260.596,A -85,B 0,C 180,E1 -3244.017,E2 -3244.017} C_VEL
LIN {X 0,Y 551.88,Z 254.519,A -85,B 0,C 180,E1 -3244.931,E2 -3244.931} C_VEL
LIN {X 0,Y 551.838,Z 248.243,A -85,B 0,C 180,E1 -3245.664,E2 -3245.664} C_VEL
LIN {X 0,Y 551.967,Z 240.023,A -85,B 0,C 180,E1 -3246.388,E2 -3246.388} C_VEL
LIN {X 0,Y 552.04,Z 231.681,A -85,B 0,C 180,E1 -3246.946,E2 -3246.946} C_VEL
LIN {X 0,Y 552.208,Z 222.05,A -85,B 0,C 180,E1 -3247.404,E2 -3247.404} C_VEL
LIN {X 0,Y 551.734,Z 214.348,A -85,B 0,C 180,E1 -3247.686,E2 -3247.686} C_VEL
LIN {X 0,Y 551.795,Z 204.948,A -85,B 0,C 180,E1 -3250.643,E2 -3250.643} C_VEL
LIN {X 0,Y 551.894,Z 195.571,A -85,B 0,C 180,E1 -3253.626,E2 -3253.626} C_VEL
LIN {X 0,Y 552.001,Z 186.217,A -85,B 0,C 180,E1 -3256.647,E2 -3256.647} C_VEL
LIN {X 0,Y 552.076,Z 177.081,A -85,B 0,C 180,E1 -3259.603,E2 -3259.603} C_VEL
LIN {X 0,Y 552.151,Z 168.338,A -85,B 0,C 180,E1 -3262.449,E2 -3262.449} C_VEL
LIN {X 0,Y 552.203,Z 159.447,A -85,B 0,C 180,E1 -3265.359,E2 -3265.359} C_VEL
LIN {X 0,Y 552.344,Z 152.478,A -85,B 0,C 180,E1 -3267.673,E2 -3267.673} C_VEL
LIN {X 0,Y 552.415,Z 145.239,A -85,B 0,C 180,E1 -3270.103,E2 -3270.103} C_VEL
LIN {X 0,Y 552.135,Z 143.713,A -85,B 0,C 180,E1 -3270.713,E2 -3270.713} C_VEL
LIN {X 0,Y 552.112,Z 143.714,A -85,B 0,C 180,E1 -3273.186,E2 -3273.186} C_VEL
LIN {X 0,Y 552.091,Z 143.718,A -85,B 0,C 180,E1 -3275.843,E2 -3275.843} C_VEL
LIN {X 0,Y 552.122,Z 143.713,A -85,B 0,C 180,E1 -3278.589,E2 -3278.589} C_VEL
LIN {X 0,Y 552.126,Z 143.714,A -85,B 0,C 180,E1 -3281.446,E2 -3281.446} C_VEL
LIN {X 0,Y 552.097,Z 143.717,A -85,B 0,C 180,E1 -3284.531,E2 -3284.531} C_VEL
LIN {X 0,Y 552.136,Z 143.711,A -85,B 0,C 180,E1 -3287.584,E2 -3287.584} C_VEL
LIN {X 0,Y 552.134,Z 143.711,A -85,B 0,C 180,E1 -3290.472,E2 -3290.472} C_VEL
LIN {X 0,Y 552.112,Z 143.716,A -85,B 0,C 180,E1 -3293.317,E2 -3293.317} C_VEL
LIN {X 0,Y 552.111,Z 143.714,A -85,B 0,C 180,E1 -3295.937,E2 -3295.937} C_VEL
LIN {X 0,Y 552.126,Z 143.715,A -85,B 0,C 180,E1 -3298.54,E2 -3298.54} C_VEL
LIN {X 0,Y 552.111,Z 143.719,A -85,B 0,C 180,E1 -3301.441,E2 -3301.441} C_VEL
LIN {X 0,Y 552.148,Z 143.848,A -85,B 0,C 180,E1 -3301.714,E2 -3301.714} C_VEL
LIN {X 0,Y 553.351,Z 150.133,A -85,B 0,C 180,E1 -3303.212,E2 -3303.212} C_VEL
LIN {X 0,Y 553.214,Z 157.544,A -85,B 0,C 180,E1 -3304.812,E2 -3304.812} C_VEL
LIN {X 0,Y 552.851,Z 171.152,A -85,B 0,C 180,E1 -3307.581,E2 -3307.581} C_VEL
LIN {X 0,Y 552.552,Z 185.951,A -85,B 0,C 180,E1 -3310.472,E2 -3310.472} C_VEL
LIN {X 0,Y 552.344,Z 200.392,A -85,B 0,C 180,E1 -3313.173,E2 -3313.173} C_VEL
LIN {X 0,Y 552.161,Z 217.756,A -85,B 0,C 180,E1 -3316.38,E2 -3316.38} C_VEL
LIN {X 0,Y 552.106,Z 221.014,A -85,B 0,C 180,E1 -3316.964,E2 -3316.964} C_VEL
LIN {X 0,Y 553.128,Z 228.037,A -85,B 0,C 180,E1 -3317.105,E2 -3317.105} C_VEL
LIN {X 0,Y 553.003,Z 240.946,A -85,B 0,C 180,E1 -3317.429,E2 -3317.429} C_VEL
LIN {X 0,Y 552.812,Z 253.465,A -85,B 0,C 180,E1 -3317.89,E2 -3317.89} C_VEL
LIN {X 0,Y 552.635,Z 265.156,A -85,B 0,C 180,E1 -3318.477,E2 -3318.477} C_VEL
LIN {X 0,Y 552.491,Z 276.179,A -85,B 0,C 180,E1 -3319.185,E2 -3319.185} C_VEL
LIN {X 0,Y 552.301,Z 286.593,A -85,B 0,C 180,E1 -3320.015,E2 -3320.015} C_VEL
LIN {X 0,Y 552.132,Z 295.103,A -85,B 0,C 180,E1 -3320.844,E2 -3320.844} C_VEL
LIN {X 0,Y 552.013,Z 302.952,A -85,B 0,C 180,E1 -3321.764,E2 -3321.764} C_VEL
LIN {X 0,Y 551.891,Z 310.615,A -85,B 0,C 180,E1 -3322.867,E2 -3322.867} C_VEL
LIN {X 0,Y 551.868,Z 317.674,A -85,B 0,C 180,E1 -3324.152,E2 -3324.152} C_VEL
LIN {X 0,Y 551.725,Z 322.369,A -85,B 0,C 180,E1 -3325.249,E2 -3325.249} C_VEL
LIN {X 0,Y 551.751,Z 325.955,A -85,B 0,C 180,E1 -3326.347,E2 -3326.347} C_VEL
LIN {X 0,Y 551.724,Z 327.805,A -85,B 0,C 180,E1 -3327.078,E2 -3327.078} C_VEL
LIN {X 0,Y 551.645,Z 330.182,A -85,B 0,C 180,E1 -3328.539,E2 -3328.539} C_VEL
LIN {X 0,Y 551.64,Z 331,A -85,B 0,C 180,E1 -3329.999,E2 -3329.999} C_VEL
LIN {X 0,Y 551.645,Z 330.185,A -85,B 0,C 180,E1 -3331.459,E2 -3331.459} C_VEL
LIN {X 0,Y 551.723,Z 327.813,A -85,B 0,C 180,E1 -3332.919,E2 -3332.919} C_VEL
LIN {X 0,Y 551.763,Z 324.899,A -85,B 0,C 180,E1 -3334.016,E2 -3334.016} C_VEL
LIN {X 0,Y 551.723,Z 320.954,A -85,B 0,C 180,E1 -3335.115,E2 -3335.115} C_VEL
LIN {X 0,Y 551.815,Z 315.126,A -85,B 0,C 180,E1 -3336.353,E2 -3336.353} C_VEL
LIN {X 0,Y 551.925,Z 308.244,A -85,B 0,C 180,E1 -3337.498,E2 -3337.498} C_VEL
LIN {X 0,Y 552.081,Z 300.003,A -85,B 0,C 180,E1 -3338.601,E2 -3338.601} C_VEL
LIN {X 0,Y 552.2,Z 291.553,A -85,B 0,C 180,E1 -3339.522,E2 -3339.522} C_VEL
LIN {X 0,Y 552.408,Z 281.108,A -85,B 0,C 180,E1 -3340.444,E2 -3340.444} C_VEL
LIN {X 0,Y 552.591,Z 270.296,A -85,B 0,C 180,E1 -3341.213,E2 -3341.213} C_VEL
LIN {X 0,Y 552.717,Z 259.43,A -85,B 0,C 180,E1 -3341.83,E2 -3341.83} C_VEL
LIN {X 0,Y 552.907,Z 247.8,A -85,B 0,C 180,E1 -3342.338,E2 -3342.338} C_VEL
LIN {X 0,Y 553.045,Z 234.396,A -85,B 0,C 180,E1 -3342.755,E2 -3342.755} C_VEL
LIN {X 0,Y 552.913,Z 226.238,A -85,B 0,C 180,E1 -3342.936,E2 -3342.936} C_VEL
LIN {X 0,Y 552.112,Z 220.818,A -85,B 0,C 180,E1 -3343.057,E2 -3343.057} C_VEL
LIN {X 0,Y 552.291,Z 204.494,A -85,B 0,C 180,E1 -3346.066,E2 -3346.066} C_VEL
LIN {X 0,Y 552.446,Z 190.177,A -85,B 0,C 180,E1 -3348.735,E2 -3348.735} C_VEL
LIN {X 0,Y 552.717,Z 177.237,A -85,B 0,C 180,E1 -3351.245,E2 -3351.245} C_VEL
LIN {X 0,Y 553.083,Z 162.264,A -85,B 0,C 180,E1 -3354.191,E2 -3354.191} C_VEL
LIN {X 0,Y 553.26,Z 151.177,A -85,B 0,C 180,E1 -3356.396,E2 -3356.396} C_VEL
LIN {X 0,Y 552.852,Z 147.158,A -85,B 0,C 180,E1 -3357.233,E2 -3357.233} C_VEL
LIN {X 0,Y 552.133,Z 143.711,A -85,B 0,C 180,E1 -3358.044,E2 -3358.044} C_VEL
LIN {X 0,Y 552.087,Z 143.719,A -85,B 0,C 180,E1 -3360.608,E2 -3360.608} C_VEL
LIN {X 0,Y 552.118,Z 143.709,A -85,B 0,C 180,E1 -3363.184,E2 -3363.184} C_VEL
LIN {X 0,Y 552.109,Z 143.717,A -85,B 0,C 180,E1 -3365.84,E2 -3365.84} C_VEL
LIN {X 0,Y 552.114,Z 143.715,A -85,B 0,C 180,E1 -3369.06,E2 -3369.06} C_VEL
LIN {X 0,Y 552.1,Z 143.71,A -85,B 0,C 180,E1 -3371.446,E2 -3371.446} C_VEL
LIN {X 0,Y 552.084,Z 143.715,A -85,B 0,C 180,E1 -3374.53,E2 -3374.53} C_VEL
LIN {X 0,Y 552.121,Z 143.714,A -85,B 0,C 180,E1 -3377.583,E2 -3377.583} C_VEL
LIN {X 0,Y 552.125,Z 143.71,A -85,B 0,C 180,E1 -3380.472,E2 -3380.472} C_VEL
LIN {X 0,Y 552.086,Z 143.712,A -85,B 0,C 180,E1 -3383.317,E2 -3383.317} C_VEL
LIN {X 0,Y 552.111,Z 143.716,A -85,B 0,C 180,E1 -3385.938,E2 -3385.938} C_VEL
LIN {X 0,Y 552.106,Z 143.71,A -85,B 0,C 180,E1 -3388.54,E2 -3388.54} C_VEL
LIN {X 0,Y 552.115,Z 143.711,A -85,B 0,C 180,E1 -3391.436,E2 -3391.436} C_VEL
LIN {X 0,Y 552.125,Z 143.713,A -85,B 0,C 180,E1 -3394.355,E2 -3394.355} C_VEL
LIN {X 0,Y 552.081,Z 143.712,A -85,B 0,C 180,E1 -3396.757,E2 -3396.757} C_VEL
LIN {X 0,Y 552.107,Z 143.713,A -85,B 0,C 180,E1 -3399.119,E2 -3399.119} C_VEL
LIN {X 0,Y 552.12,Z 143.71,A -85,B 0,C 180,E1 -3401.444,E2 -3401.444} C_VEL
LIN {X 0,Y 552.11,Z 143.71,A -85,B 0,C 180,E1 -3403.737,E2 -3403.737} C_VEL
LIN {X 0,Y 552.127,Z 143.714,A -85,B 0,C 180,E1 -3406.004,E2 -3406.004} C_VEL
LIN {X 0,Y 552.142,Z 143.707,A -85,B 0,C 180,E1 -3408.993,E2 -3408.993} C_VEL
LIN {X 0,Y 552.139,Z 143.706,A -85,B 0,C 180,E1 -3411.951,E2 -3411.951} C_VEL
LIN {X 0,Y 552.22,Z 143.698,A -85,B 0,C 180,E1 -3414.889,E2 -3414.889} C_VEL
LIN {X 0,Y 552.212,Z 143.702,A -85,B 0,C 180,E1 -3417.812,E2 -3417.812} C_VEL
LIN {X 0,Y 552.227,Z 143.696,A -85,B 0,C 180,E1 -3420.729,E2 -3420.729} C_VEL
LIN {X 0,Y 552.185,Z 143.706,A -85,B 0,C 180,E1 -3422.918,E2 -3422.918} C_VEL
LIN {X 0,Y 552.183,Z 143.703,A -85,B 0,C 180,E1 -3425.844,E2 -3425.844} C_VEL
LIN {X 0,Y 552.16,Z 143.704,A -85,B 0,C 180,E1 -3428.786,E2 -3428.786} C_VEL
LIN {X 0,Y 552.149,Z 143.706,A -85,B 0,C 180,E1 -3431.751,E2 -3431.751} C_VEL
LIN {X 0,Y 552.12,Z 143.712,A -85,B 0,C 180,E1 -3434.749,E2 -3434.749} C_VEL
LIN {X 0,Y 552.101,Z 143.715,A -85,B 0,C 180,E1 -3437.789,E2 -3437.789} C_VEL
LIN {X 0,Y 552.121,Z 143.71,A -85,B 0,C 180,E1 -3440.102,E2 -3440.102} C_VEL
LIN {X 0,Y 552.102,Z 143.712,A -85,B 0,C 180,E1 -3442.451,E2 -3442.451} C_VEL
LIN {X 0,Y 552.122,Z 143.708,A -85,B 0,C 180,E1 -3445.347,E2 -3445.347} C_VEL
LIN {X 0,Y 552.063,Z 143.721,A -85,B 0,C 180,E1 -3448.101,E2 -3448.101} C_VEL
LIN {X 0,Y 552.096,Z 143.711,A -85,B 0,C 180,E1 -3450.633,E2 -3450.633} C_VEL
LIN {X 0,Y 552.117,Z 143.714,A -85,B 0,C 180,E1 -3453.186,E2 -3453.186} C_VEL
LIN {X 0,Y 552.113,Z 143.71,A -85,B 0,C 180,E1 -3453.813,E2 -3453.813} C_VEL
LIN {X 0,Y 551.48,Z 143.793,A -85,B 0,C 180,E1 -3454.422,E2 -3454.422} C_VEL
LIN {X 0,Y 548.653,Z 144.143,A -85,B 0,C 180,E1 -3455.41,E2 -3455.41} C_VEL
LIN {X 0,Y 546.226,Z 144.447,A -85,B 0,C 180,E1 -3456.205,E2 -3456.205} C_VEL
LIN {X 0,Y 545.154,Z 144.578,A -85,B 0,C 180,E1 -3456.819,E2 -3456.819} C_VEL
LIN {X 0,Y 545.051,Z 144.589,A -85,B 0,C 180,E1 -3457.027,E2 -3457.027} C_VEL
LIN {X 0,Y 545.053,Z 144.59,A -85,B 0,C 180,E1 -3460.144,E2 -3460.144} C_VEL
LIN {X 0,Y 545.076,Z 144.591,A -85,B 0,C 180,E1 -3463.107,E2 -3463.107} C_VEL
LIN {X 0,Y 545.056,Z 144.592,A -85,B 0,C 180,E1 -3466.226,E2 -3466.226} C_VEL
LIN {X 0,Y 545.089,Z 144.585,A -85,B 0,C 180,E1 -3468.888,E2 -3468.888} C_VEL
LIN {X 0,Y 545.039,Z 144.593,A -85,B 0,C 180,E1 -3471.764,E2 -3471.764} C_VEL
LIN {X 0,Y 545.023,Z 144.594,A -85,B 0,C 180,E1 -3474.532,E2 -3474.532} C_VEL
LIN {X 0,Y 545.076,Z 144.586,A -85,B 0,C 180,E1 -3477.214,E2 -3477.214} C_VEL
LIN {X 0,Y 545.097,Z 144.589,A -85,B 0,C 180,E1 -3479.814,E2 -3479.814} C_VEL
LIN {X 0,Y 545.09,Z 144.586,A -85,B 0,C 180,E1 -3482.828,E2 -3482.828} C_VEL
LIN {X 0,Y 545.015,Z 144.593,A -85,B 0,C 180,E1 -3485.631,E2 -3485.631} C_VEL
LIN {X 0,Y 545.062,Z 144.589,A -85,B 0,C 180,E1 -3488.838,E2 -3488.838} C_VEL
LIN {X 0,Y 545.079,Z 144.587,A -85,B 0,C 180,E1 -3491.197,E2 -3491.197} C_VEL
LIN {X 0,Y 545.071,Z 144.591,A -85,B 0,C 180,E1 -3493.523,E2 -3493.523} C_VEL
LIN {X 0,Y 545.079,Z 144.585,A -85,B 0,C 180,E1 -3495.821,E2 -3495.821} C_VEL
LIN {X 0,Y 545.115,Z 144.582,A -85,B 0,C 180,E1 -3498.851,E2 -3498.851} C_VEL
LIN {X 0,Y 545.125,Z 144.585,A -85,B 0,C 180,E1 -3501.848,E2 -3501.848} C_VEL
LIN {X 0,Y 545.204,Z 144.574,A -85,B 0,C 180,E1 -3504.824,E2 -3504.824} C_VEL
LIN {X 0,Y 545.197,Z 144.571,A -85,B 0,C 180,E1 -3507.785,E2 -3507.785} C_VEL
LIN {X 0,Y 545.193,Z 144.576,A -85,B 0,C 180,E1 -3510.001,E2 -3510.001} C_VEL
LIN {X 0,Y 545.163,Z 144.576,A -85,B 0,C 180,E1 -3512.957,E2 -3512.957} C_VEL
LIN {X 0,Y 545.174,Z 144.574,A -85,B 0,C 180,E1 -3515.921,E2 -3515.921} C_VEL
LIN {X 0,Y 545.113,Z 144.583,A -85,B 0,C 180,E1 -3518.901,E2 -3518.901} C_VEL
LIN {X 0,Y 545.097,Z 144.589,A -85,B 0,C 180,E1 -3521.906,E2 -3521.906} C_VEL
LIN {X 0,Y 545.081,Z 144.588,A -85,B 0,C 180,E1 -3524.945,E2 -3524.945} C_VEL
LIN {X 0,Y 545.076,Z 144.587,A -85,B 0,C 180,E1 -3528.027,E2 -3528.027} C_VEL
LIN {X 0,Y 545.097,Z 144.588,A -85,B 0,C 180,E1 -3530.373,E2 -3530.373} C_VEL
LIN {X 0,Y 545.074,Z 144.592,A -85,B 0,C 180,E1 -3533.561,E2 -3533.561} C_VEL
LIN {X 0,Y 545.042,Z 144.589,A -85,B 0,C 180,E1 -3536.003,E2 -3536.003} C_VEL
LIN {X 0,Y 545.051,Z 144.595,A -85,B 0,C 180,E1 -3538.74,E2 -3538.74} C_VEL
LIN {X 0,Y 545.063,Z 144.59,A -85,B 0,C 180,E1 -3541.679,E2 -3541.679} C_VEL
LIN {X 0,Y 545.064,Z 144.588,A -85,B 0,C 180,E1 -3544.565,E2 -3544.565} C_VEL
LIN {X 0,Y 545.024,Z 144.595,A -85,B 0,C 180,E1 -3547.306,E2 -3547.306} C_VEL
LIN {X 0,Y 545.058,Z 144.591,A -85,B 0,C 180,E1 -3550.144,E2 -3550.144} C_VEL
LIN {X 0,Y 545.05,Z 144.59,A -85,B 0,C 180,E1 -3553.11,E2 -3553.11} C_VEL
LIN {X 0,Y 545.054,Z 144.589,A -85,B 0,C 180,E1 -3556.227,E2 -3556.227} C_VEL
LIN {X 0,Y 545.085,Z 144.589,A -85,B 0,C 180,E1 -3558.886,E2 -3558.886} C_VEL
LIN {X 0,Y 545.043,Z 144.592,A -85,B 0,C 180,E1 -3561.866,E2 -3561.866} C_VEL
LIN {X 0,Y 545.033,Z 144.591,A -85,B 0,C 180,E1 -3564.531,E2 -3564.531} C_VEL
LIN {X 0,Y 545.069,Z 144.593,A -85,B 0,C 180,E1 -3567.212,E2 -3567.212} C_VEL
LIN {X 0,Y 545.097,Z 144.601,A -85,B 0,C 180,E1 -3569.265,E2 -3569.265} C_VEL
LIN {X 0,Y 545.428,Z 148.604,A -85,B 0,C 180,E1 -3570.683,E2 -3570.683} C_VEL
LIN {X 0,Y 545.287,Z 157.065,A -85,B 0,C 180,E1 -3573.599,E2 -3573.599} C_VEL
LIN {X 0,Y 545.126,Z 165.518,A -85,B 0,C 180,E1 -3576.443,E2 -3576.443} C_VEL
LIN {X 0,Y 545.039,Z 173.97,A -85,B 0,C 180,E1 -3579.231,E2 -3579.231} C_VEL
LIN {X 0,Y 544.957,Z 182.392,A -85,B 0,C 180,E1 -3581.97,E2 -3581.97} C_VEL
LIN {X 0,Y 544.881,Z 191.774,A -85,B 0,C 180,E1 -3585.051,E2 -3585.051} C_VEL
LIN {X 0,Y 544.739,Z 201.172,A -85,B 0,C 180,E1 -3588.087,E2 -3588.087} C_VEL
LIN {X 0,Y 544.692,Z 209.408,A -85,B 0,C 180,E1 -3590.719,E2 -3590.719} C_VEL
LIN {X 0,Y 544.66,Z 214.552,A -85,B 0,C 180,E1 -3592.307,E2 -3592.307} C_VEL
LIN {X 0,Y 545.162,Z 222.678,A -85,B 0,C 180,E1 -3592.593,E2 -3592.593} C_VEL
LIN {X 0,Y 545.044,Z 232.308,A -85,B 0,C 180,E1 -3593.069,E2 -3593.069} C_VEL
LIN {X 0,Y 544.951,Z 240.304,A -85,B 0,C 180,E1 -3593.613,E2 -3593.613} C_VEL
LIN {X 0,Y 544.793,Z 247.729,A -85,B 0,C 180,E1 -3594.262,E2 -3594.262} C_VEL
LIN {X 0,Y 544.828,Z 254.185,A -85,B 0,C 180,E1 -3595.005,E2 -3595.005} C_VEL
LIN {X 0,Y 544.739,Z 259.29,A -85,B 0,C 180,E1 -3595.746,E2 -3595.746} C_VEL
LIN {X 0,Y 544.713,Z 264.161,A -85,B 0,C 180,E1 -3596.672,E2 -3596.672} C_VEL
LIN {X 0,Y 544.59,Z 268.156,A -85,B 0,C 180,E1 -3597.781,E2 -3597.781} C_VEL
LIN {X 0,Y 544.556,Z 269.889,A -85,B 0,C 180,E1 -3598.521,E2 -3598.521} C_VEL
LIN {X 0,Y 544.55,Z 270.928,A -85,B 0,C 180,E1 -3599.261,E2 -3599.261} C_VEL
LIN {X 0,Y 544.548,Z 271.302,A -85,B 0,C 180,E1 -3600,E2 -3600} C_VEL
LIN {X 0,Y 544.549,Z 271.02,A -85,B 0,C 180,E1 -3600.74,E2 -3600.74} C_VEL
LIN {X 0,Y 544.558,Z 270.076,A -85,B 0,C 180,E1 -3601.479,E2 -3601.479} C_VEL
LIN {X 0,Y 544.59,Z 268.446,A -85,B 0,C 180,E1 -3602.219,E2 -3602.219} C_VEL
LIN {X 0,Y 544.713,Z 264.57,A -85,B 0,C 180,E1 -3603.329,E2 -3603.329} C_VEL
LIN {X 0,Y 544.737,Z 259.916,A -85,B 0,C 180,E1 -3604.254,E2 -3604.254} C_VEL
LIN {X 0,Y 544.811,Z 254.948,A -85,B 0,C 180,E1 -3604.995,E2 -3604.995} C_VEL
LIN {X 0,Y 544.788,Z 248.688,A -85,B 0,C 180,E1 -3605.738,E2 -3605.738} C_VEL
LIN {X 0,Y 544.93,Z 241.731,A -85,B 0,C 180,E1 -3606.379,E2 -3606.379} C_VEL
LIN {X 0,Y 544.999,Z 234.074,A -85,B 0,C 180,E1 -3606.924,E2 -3606.924} C_VEL
LIN {X 0,Y 545.165,Z 225.133,A -85,B 0,C 180,E1 -3607.407,E2 -3607.407} C_VEL
LIN {X 0,Y 544.89,Z 216.576,A -85,B 0,C 180,E1 -3607.737,E2 -3607.737} C_VEL
LIN {X 0,Y 544.671,Z 214.379,A -85,B 0,C 180,E1 -3607.833,E2 -3607.833} C_VEL
LIN {X 0,Y 544.733,Z 205.057,A -85,B 0,C 180,E1 -3610.782,E2 -3610.782} C_VEL
LIN {X 0,Y 544.851,Z 195.68,A -85,B 0,C 180,E1 -3613.806,E2 -3613.806} C_VEL
LIN {X 0,Y 544.932,Z 186.328,A -85,B 0,C 180,E1 -3616.869,E2 -3616.869} C_VEL
LIN {X 0,Y 545.026,Z 177.561,A -85,B 0,C 180,E1 -3619.724,E2 -3619.724} C_VEL
LIN {X 0,Y 545.117,Z 168.363,A -85,B 0,C 180,E1 -3622.754,E2 -3622.754} C_VEL
LIN {X 0,Y 545.216,Z 160.05,A -85,B 0,C 180,E1 -3625.534,E2 -3625.534} C_VEL
LIN {X 0,Y 545.354,Z 152.563,A -85,B 0,C 180,E1 -3628.059,E2 -3628.059} C_VEL
LIN {X 0,Y 545.409,Z 146.402,A -85,B 0,C 180,E1 -3630.169,E2 -3630.169} C_VEL
LIN {X 0,Y 545.103,Z 144.589,A -85,B 0,C 180,E1 -3630.84,E2 -3630.84} C_VEL
LIN {X 0,Y 545.055,Z 144.595,A -85,B 0,C 180,E1 -3633.673,E2 -3633.673} C_VEL
LIN {X 0,Y 545.076,Z 144.592,A -85,B 0,C 180,E1 -3636.926,E2 -3636.926} C_VEL
LIN {X 0,Y 545.071,Z 144.592,A -85,B 0,C 180,E1 -3640.142,E2 -3640.142} C_VEL
LIN {X 0,Y 545.084,Z 144.589,A -85,B 0,C 180,E1 -3643.106,E2 -3643.106} C_VEL
LIN {X 0,Y 545.073,Z 144.59,A -85,B 0,C 180,E1 -3646.224,E2 -3646.224} C_VEL
LIN {X 0,Y 545.088,Z 144.59,A -85,B 0,C 180,E1 -3648.885,E2 -3648.885} C_VEL
LIN {X 0,Y 545.055,Z 144.593,A -85,B 0,C 180,E1 -3651.762,E2 -3651.762} C_VEL
LIN {X 0,Y 545.044,Z 144.596,A -85,B 0,C 180,E1 -3654.531,E2 -3654.531} C_VEL
LIN {X 0,Y 545.071,Z 144.592,A -85,B 0,C 180,E1 -3657.211,E2 -3657.211} C_VEL
LIN {X 0,Y 545.069,Z 144.597,A -85,B 0,C 180,E1 -3659.81,E2 -3659.81} C_VEL
LIN {X 0,Y 545.101,Z 144.746,A -85,B 0,C 180,E1 -3661.418,E2 -3661.418} C_VEL
LIN {X 0,Y 546.335,Z 150.834,A -85,B 0,C 180,E1 -3662.933,E2 -3662.933} C_VEL
LIN {X 0,Y 546.426,Z 156.479,A -85,B 0,C 180,E1 -3664.201,E2 -3664.201} C_VEL
LIN {X 0,Y 545.927,Z 169.175,A -85,B 0,C 180,E1 -3666.88,E2 -3666.88} C_VEL
LIN {X 0,Y 545.595,Z 184.408,A -85,B 0,C 180,E1 -3669.937,E2 -3669.937} C_VEL
LIN {X 0,Y 545.342,Z 199.242,A -85,B 0,C 180,E1 -3672.757,E2 -3672.757} C_VEL
LIN {X 0,Y 545.103,Z 213.976,A -85,B 0,C 180,E1 -3675.518,E2 -3675.518} C_VEL
LIN {X 0,Y 545.068,Z 221.057,A -85,B 0,C 180,E1 -3676.828,E2 -3676.828} C_VEL
LIN {X 0,Y 546.138,Z 228.992,A -85,B 0,C 180,E1 -3676.984,E2 -3676.984} C_VEL
LIN {X 0,Y 546.031,Z 241.662,A -85,B 0,C 180,E1 -3677.313,E2 -3677.313} C_VEL
LIN {X 0,Y 545.824,Z 254.028,A -85,B 0,C 180,E1 -3677.78,E2 -3677.78} C_VEL
LIN {X 0,Y 545.635,Z 265.723,A -85,B 0,C 180,E1 -3678.377,E2 -3678.377} C_VEL
LIN {X 0,Y 545.45,Z 277.367,A -85,B 0,C 180,E1 -3679.137,E2 -3679.137} C_VEL
LIN {X 0,Y 545.276,Z 287.629,A -85,B 0,C 180,E1 -3679.978,E2 -3679.978} C_VEL
LIN {X 0,Y 545.082,Z 296.776,A -85,B 0,C 180,E1 -3680.911,E2 -3680.911} C_VEL
LIN {X 0,Y 544.917,Z 305.68,A -85,B 0,C 180,E1 -3682.029,E2 -3682.029} C_VEL
LIN {X 0,Y 544.786,Z 312.842,A -85,B 0,C 180,E1 -3683.146,E2 -3683.146} C_VEL
LIN {X 0,Y 544.741,Z 319.361,A -85,B 0,C 180,E1 -3684.446,E2 -3684.446} C_VEL
LIN {X 0,Y 544.66,Z 323.673,A -85,B 0,C 180,E1 -3685.559,E2 -3685.559} C_VEL
LIN {X 0,Y 544.669,Z 325.955,A -85,B 0,C 180,E1 -3686.3,E2 -3686.3} C_VEL
LIN {X 0,Y 544.651,Z 327.804,A -85,B 0,C 180,E1 -3687.04,E2 -3687.04} C_VEL
LIN {X 0,Y 544.546,Z 330.181,A -85,B 0,C 180,E1 -3688.52,E2 -3688.52} C_VEL
LIN {X 0,Y 544.541,Z 331,A -85,B 0,C 180,E1 -3689.999,E2 -3689.999} C_VEL
LIN {X 0,Y 544.546,Z 330.185,A -85,B 0,C 180,E1 -3691.478,E2 -3691.478} C_VEL
LIN {X 0,Y 544.65,Z 327.813,A -85,B 0,C 180,E1 -3692.957,E2 -3692.957} C_VEL
LIN {X 0,Y 544.683,Z 324.899,A -85,B 0,C 180,E1 -3694.068,E2 -3694.068} C_VEL
LIN {X 0,Y 544.653,Z 320.953,A -85,B 0,C 180,E1 -3695.181,E2 -3695.181} C_VEL
LIN {X 0,Y 544.729,Z 315.645,A -85,B 0,C 180,E1 -3696.339,E2 -3696.339} C_VEL
LIN {X 0,Y 544.835,Z 309.474,A -85,B 0,C 180,E1 -3697.41,E2 -3697.41} C_VEL
LIN {X 0,Y 545.005,Z 301.487,A -85,B 0,C 180,E1 -3698.527,E2 -3698.527} C_VEL
LIN {X 0,Y 545.141,Z 293.345,A -85,B 0,C 180,E1 -3699.46,E2 -3699.46} C_VEL
LIN {X 0,Y 545.359,Z 283.382,A -85,B 0,C 180,E1 -3700.393,E2 -3700.393} C_VEL
LIN {X 0,Y 545.554,Z 272.455,A -85,B 0,C 180,E1 -3701.207,E2 -3701.207} C_VEL
LIN {X 0,Y 545.702,Z 260.886,A -85,B 0,C 180,E1 -3701.89,E2 -3701.89} C_VEL
LIN {X 0,Y 545.915,Z 248.505,A -85,B 0,C 180,E1 -3702.451,E2 -3702.451} C_VEL
LIN {X 0,Y 546.083,Z 235.344,A -85,B 0,C 180,E1 -3702.873,E2 -3702.873} C_VEL
LIN {X 0,Y 545.948,Z 226.963,A -85,B 0,C 180,E1 -3703.065,E2 -3703.065} C_VEL
LIN {X 0,Y 545.054,Z 220.96,A -85,B 0,C 180,E1 -3703.182,E2 -3703.182} C_VEL
LIN {X 0,Y 545.264,Z 204.368,A -85,B 0,C 180,E1 -3706.279,E2 -3706.279} C_VEL
LIN {X 0,Y 545.459,Z 190.05,A -85,B 0,C 180,E1 -3708.984,E2 -3708.984} C_VEL
LIN {X 0,Y 545.878,Z 174.685,A -85,B 0,C 180,E1 -3712.031,E2 -3712.031} C_VEL
LIN {X 0,Y 546.227,Z 159.291,A -85,B 0,C 180,E1 -3715.123,E2 -3715.123} C_VEL
LIN {X 0,Y 546.283,Z 151.229,A -85,B 0,C 180,E1 -3716.76,E2 -3716.76} C_VEL
LIN {X 0,Y 545.078,Z 144.591,A -85,B 0,C 180,E1 -3718.256,E2 -3718.256} C_VEL
LIN {X 0,Y 545.057,Z 144.592,A -85,B 0,C 180,E1 -3721.047,E2 -3721.047} C_VEL
LIN {X 0,Y 545.066,Z 144.589,A -85,B 0,C 180,E1 -3723.67,E2 -3723.67} C_VEL
LIN {X 0,Y 545.05,Z 144.59,A -85,B 0,C 180,E1 -3726.378,E2 -3726.378} C_VEL
LIN {X 0,Y 545.094,Z 144.588,A -85,B 0,C 180,E1 -3729.322,E2 -3729.322} C_VEL
LIN {X 0,Y 545.052,Z 144.59,A -85,B 0,C 180,E1 -3732.103,E2 -3732.103} C_VEL
LIN {X 0,Y 545.053,Z 144.589,A -85,B 0,C 180,E1 -3735.166,E2 -3735.166} C_VEL
LIN {X 0,Y 545.074,Z 144.589,A -85,B 0,C 180,E1 -3737.896,E2 -3737.896} C_VEL
LIN {X 0,Y 545.096,Z 144.588,A -85,B 0,C 180,E1 -3740.674,E2 -3740.674} C_VEL
LIN {X 0,Y 545.02,Z 144.593,A -85,B 0,C 180,E1 -3743.618,E2 -3743.618} C_VEL
LIN {X 0,Y 545.054,Z 144.59,A -85,B 0,C 180,E1 -3746.327,E2 -3746.327} C_VEL
LIN {X 0,Y 545.059,Z 144.591,A -85,B 0,C 180,E1 -3748.952,E2 -3748.952} C_VEL
LIN {X 0,Y 545.093,Z 144.585,A -85,B 0,C 180,E1 -3751.507,E2 -3751.507} C_VEL
LIN {X 0,Y 545.087,Z 144.588,A -85,B 0,C 180,E1 -3754.489,E2 -3754.489} C_VEL
LIN {X 0,Y 545.02,Z 144.594,A -85,B 0,C 180,E1 -3757.241,E2 -3757.241} C_VEL
LIN {X 0,Y 545.106,Z 144.583,A -85,B 0,C 180,E1 -3760.414,E2 -3760.414} C_VEL
LIN {X 0,Y 545.066,Z 144.587,A -85,B 0,C 180,E1 -3763.521,E2 -3763.521} C_VEL
LIN {X 0,Y 545.084,Z 144.589,A -85,B 0,C 180,E1 -3765.82,E2 -3765.82} C_VEL
LIN {X 0,Y 545.098,Z 144.583,A -85,B 0,C 180,E1 -3768.849,E2 -3768.849} C_VEL
LIN {X 0,Y 545.11,Z 144.581,A -85,B 0,C 180,E1 -3771.847,E2 -3771.847} C_VEL
LIN {X 0,Y 545.195,Z 144.574,A -85,B 0,C 180,E1 -3774.823,E2 -3774.823} C_VEL
LIN {X 0,Y 545.184,Z 144.578,A -85,B 0,C 180,E1 -3777.784,E2 -3777.784} C_VEL
LIN {X 0,Y 545.197,Z 144.572,A -85,B 0,C 180,E1 -3780.739,E2 -3780.739} C_VEL
LIN {X 0,Y 545.151,Z 144.581,A -85,B 0,C 180,E1 -3782.956,E2 -3782.956} C_VEL
LIN {X 0,Y 545.155,Z 144.579,A -85,B 0,C 180,E1 -3785.92,E2 -3785.92} C_VEL
LIN {X 0,Y 545.117,Z 144.581,A -85,B 0,C 180,E1 -3788.9,E2 -3788.9} C_VEL
LIN {X 0,Y 545.121,Z 144.581,A -85,B 0,C 180,E1 -3791.904,E2 -3791.904} C_VEL
LIN {X 0,Y 545.069,Z 144.588,A -85,B 0,C 180,E1 -3794.944,E2 -3794.944} C_VEL
LIN {X 0,Y 545.069,Z 144.593,A -85,B 0,C 180,E1 -3798.026,E2 -3798.026} C_VEL
LIN {X 0,Y 545.086,Z 144.585,A -85,B 0,C 180,E1 -3800.372,E2 -3800.372} C_VEL
LIN {X 0,Y 545.101,Z 144.584,A -85,B 0,C 180,E1 -3803.558,E2 -3803.558} C_VEL
LIN {X 0,Y 545.059,Z 144.59,A -85,B 0,C 180,E1 -3806.002,E2 -3806.002} C_VEL
LIN {X 0,Y 545.055,Z 144.588,A -85,B 0,C 180,E1 -3808.745,E2 -3808.745} C_VEL
LIN {X 0,Y 545.056,Z 144.591,A -85,B 0,C 180,E1 -3811.049,E2 -3811.049} C_VEL
LIN {X 0,Y 545.062,Z 144.588,A -85,B 0,C 180,E1 -3813.812,E2 -3813.812} C_VEL
LIN {X 0,Y 545.063,Z 144.588,A -85,B 0,C 180,E1 -3816.928,E2 -3816.928} C_VEL
LIN {X 0,Y 545.051,Z 144.589,A -85,B 0,C 180,E1 -3817.027,E2 -3817.027} C_VEL
LIN {X 0,Y 544.343,Z 144.68,A -85,B 0,C 180,E1 -3817.644,E2 -3817.644} C_VEL
LIN {X 0,Y 541.476,Z 145.036,A -85,B 0,C 180,E1 -3818.644,E2 -3818.644} C_VEL
LIN {X 0,Y 539.088,Z 145.335,A -85,B 0,C 180,E1 -3819.45,E2 -3819.45} C_VEL
LIN {X 0,Y 538.08,Z 145.46,A -85,B 0,C 180,E1 -3820.072,E2 -3820.072} C_VEL
LIN {X 0,Y 538.005,Z 145.467,A -85,B 0,C 180,E1 -3820.283,E2 -3820.283} C_VEL
LIN {X 0,Y 538.022,Z 145.469,A -85,B 0,C 180,E1 -3822.989,E2 -3822.989} C_VEL
LIN {X 0,Y 538.02,Z 145.466,A -85,B 0,C 180,E1 -3825.927,E2 -3825.927} C_VEL
LIN {X 0,Y 538.043,Z 145.463,A -85,B 0,C 180,E1 -3829.226,E2 -3829.226} C_VEL
LIN {X 0,Y 537.979,Z 145.47,A -85,B 0,C 180,E1 -3832.123,E2 -3832.123} C_VEL
LIN {X 0,Y 537.988,Z 145.475,A -85,B 0,C 180,E1 -3834.917,E2 -3834.917} C_VEL
LIN {X 0,Y 538.026,Z 145.465,A -85,B 0,C 180,E1 -3837.62,E2 -3837.62} C_VEL
LIN {X 0,Y 538.039,Z 145.465,A -85,B 0,C 180,E1 -3840.242,E2 -3840.242} C_VEL
LIN {X 0,Y 538.06,Z 145.461,A -85,B 0,C 180,E1 -3842.798,E2 -3842.798} C_VEL
LIN {X 0,Y 537.978,Z 145.472,A -85,B 0,C 180,E1 -3845.291,E2 -3845.291} C_VEL
LIN {X 0,Y 538.011,Z 145.469,A -85,B 0,C 180,E1 -3848.044,E2 -3848.044} C_VEL
LIN {X 0,Y 538.036,Z 145.463,A -85,B 0,C 180,E1 -3850.942,E2 -3850.942} C_VEL
LIN {X 0,Y 538.023,Z 145.47,A -85,B 0,C 180,E1 -3853.3,E2 -3853.3} C_VEL
LIN {X 0,Y 538.052,Z 145.461,A -85,B 0,C 180,E1 -3855.632,E2 -3855.632} C_VEL
LIN {X 0,Y 538.075,Z 145.46,A -85,B 0,C 180,E1 -3858.703,E2 -3858.703} C_VEL
LIN {X 0,Y 538.082,Z 145.463,A -85,B 0,C 180,E1 -3861.741,E2 -3861.741} C_VEL
LIN {X 0,Y 538.162,Z 145.45,A -85,B 0,C 180,E1 -3864.756,E2 -3864.756} C_VEL
LIN {X 0,Y 538.168,Z 145.447,A -85,B 0,C 180,E1 -3867.756,E2 -3867.756} C_VEL
LIN {X 0,Y 538.162,Z 145.452,A -85,B 0,C 180,E1 -3870.001,E2 -3870.001} C_VEL
LIN {X 0,Y 538.13,Z 145.452,A -85,B 0,C 180,E1 -3872.996,E2 -3872.996} C_VEL
LIN {X 0,Y 538.127,Z 145.452,A -85,B 0,C 180,E1 -3875.998,E2 -3875.998} C_VEL
LIN {X 0,Y 538.063,Z 145.461,A -85,B 0,C 180,E1 -3879.019,E2 -3879.019} C_VEL
LIN {X 0,Y 538.056,Z 145.464,A -85,B 0,C 180,E1 -3882.064,E2 -3882.064} C_VEL
LIN {X 0,Y 538.043,Z 145.467,A -85,B 0,C 180,E1 -3885.145,E2 -3885.145} C_VEL
LIN {X 0,Y 538.03,Z 145.467,A -85,B 0,C 180,E1 -3888.271,E2 -3888.271} C_VEL
LIN {X 0,Y 538.042,Z 145.464,A -85,B 0,C 180,E1 -3890.652,E2 -3890.652} C_VEL
LIN {X 0,Y 538.01,Z 145.469,A -85,B 0,C 180,E1 -3893.878,E2 -3893.878} C_VEL
LIN {X 0,Y 537.986,Z 145.469,A -85,B 0,C 180,E1 -3896.371,E2 -3896.371} C_VEL
LIN {X 0,Y 537.996,Z 145.471,A -85,B 0,C 180,E1 -3898.926,E2 -3898.926} C_VEL
LIN {X 0,Y 538.015,Z 145.47,A -85,B 0,C 180,E1 -3901.888,E2 -3901.888} C_VEL
LIN {X 0,Y 538.013,Z 145.466,A -85,B 0,C 180,E1 -3904.618,E2 -3904.618} C_VEL
LIN {X 0,Y 537.986,Z 145.473,A -85,B 0,C 180,E1 -3907.167,E2 -3907.167} C_VEL
LIN {X 0,Y 537.999,Z 145.467,A -85,B 0,C 180,E1 -3909.8,E2 -3909.8} C_VEL
LIN {X 0,Y 538.005,Z 145.467,A -85,B 0,C 180,E1 -3912.788,E2 -3912.788} C_VEL
LIN {X 0,Y 538.009,Z 145.47,A -85,B 0,C 180,E1 -3915.138,E2 -3915.138} C_VEL
LIN {X 0,Y 538.035,Z 145.464,A -85,B 0,C 180,E1 -3918.227,E2 -3918.227} C_VEL
LIN {X 0,Y 538.01,Z 145.465,A -85,B 0,C 180,E1 -3921.169,E2 -3921.169} C_VEL
LIN {X 0,Y 537.993,Z 145.472,A -85,B 0,C 180,E1 -3924.09,E2 -3924.09} C_VEL
LIN {X 0,Y 538.036,Z 145.465,A -85,B 0,C 180,E1 -3926.728,E2 -3926.728} C_VEL
LIN {X 0,Y 538.069,Z 145.498,A -85,B 0,C 180,E1 -3929.158,E2 -3929.158} C_VEL
LIN {X 0,Y 538.42,Z 149.726,A -85,B 0,C 180,E1 -3930.675,E2 -3930.675} C_VEL
LIN {X 0,Y 538.252,Z 158.275,A -85,B 0,C 180,E1 -3933.644,E2 -3933.644} C_VEL
LIN {X 0,Y 538.085,Z 166.727,A -85,B 0,C 180,E1 -3936.524,E2 -3936.524} C_VEL
LIN {X 0,Y 537.981,Z 176.387,A -85,B 0,C 180,E1 -3939.746,E2 -3939.746} C_VEL
LIN {X 0,Y 537.887,Z 186.001,A -85,B 0,C 180,E1 -3942.909,E2 -3942.909} C_VEL
LIN {X 0,Y 537.764,Z 195.371,A -85,B 0,C 180,E1 -3946.009,E2 -3946.009} C_VEL
LIN {X 0,Y 537.669,Z 204.775,A -85,B 0,C 180,E1 -3949.075,E2 -3949.075} C_VEL
LIN {X 0,Y 537.589,Z 214.23,A -85,B 0,C 180,E1 -3952.11,E2 -3952.11} C_VEL
LIN {X 0,Y 537.602,Z 214.654,A -85,B 0,C 180,E1 -3952.181,E2 -3952.181} C_VEL
LIN {X 0,Y 538.171,Z 223.342,A -85,B 0,C 180,E1 -3952.496,E2 -3952.496} C_VEL
LIN {X 0,Y 538.039,Z 232.578,A -85,B 0,C 180,E1 -3952.966,E2 -3952.966} C_VEL
LIN {X 0,Y 537.91,Z 241.286,A -85,B 0,C 180,E1 -3953.573,E2 -3953.573} C_VEL
LIN {X 0,Y 537.745,Z 248.093,A -85,B 0,C 180,E1 -3954.187,E2 -3954.187} C_VEL
LIN {X 0,Y 537.764,Z 254.549,A -85,B 0,C 180,E1 -3954.939,E2 -3954.939} C_VEL
LIN {X 0,Y 537.677,Z 259.654,A -85,B 0,C 180,E1 -3955.69,E2 -3955.69} C_VEL
LIN {X 0,Y 537.646,Z 264.528,A -85,B 0,C 180,E1 -3956.628,E2 -3956.628} C_VEL
LIN {X 0,Y 537.509,Z 268.534,A -85,B 0,C 180,E1 -3957.752,E2 -3957.752} C_VEL
LIN {X 0,Y 537.47,Z 270.274,A -85,B 0,C 180,E1 -3958.501,E2 -3958.501} C_VEL
LIN {X 0,Y 537.461,Z 271.318,A -85,B 0,C 180,E1 -3959.251,E2 -3959.251} C_VEL
LIN {X 0,Y 537.46,Z 271.697,A -85,B 0,C 180,E1 -3960,E2 -3960} C_VEL
LIN {X 0,Y 537.462,Z 271.419,A -85,B 0,C 180,E1 -3960.749,E2 -3960.749} C_VEL
LIN {X 0,Y 537.471,Z 270.478,A -85,B 0,C 180,E1 -3961.499,E2 -3961.499} C_VEL
LIN {X 0,Y 537.554,Z 267.729,A -85,B 0,C 180,E1 -3962.623,E2 -3962.623} C_VEL
LIN {X 0,Y 537.645,Z 264.981,A -85,B 0,C 180,E1 -3963.372,E2 -3963.372} C_VEL
LIN {X 0,Y 537.675,Z 260.325,A -85,B 0,C 180,E1 -3964.31,E2 -3964.31} C_VEL
LIN {X 0,Y 537.749,Z 255.378,A -85,B 0,C 180,E1 -3965.061,E2 -3965.061} C_VEL
LIN {X 0,Y 537.739,Z 249.131,A -85,B 0,C 180,E1 -3965.813,E2 -3965.813} C_VEL
LIN {X 0,Y 537.915,Z 241.284,A -85,B 0,C 180,E1 -3966.538,E2 -3966.538} C_VEL
LIN {X 0,Y 538.019,Z 232.847,A -85,B 0,C 180,E1 -3967.128,E2 -3967.128} C_VEL
LIN {X 0,Y 538.213,Z 222.614,A -85,B 0,C 180,E1 -3967.645,E2 -3967.645} C_VEL
LIN {X 0,Y 537.62,Z 214.596,A -85,B 0,C 180,E1 -3967.937,E2 -3967.937} C_VEL
LIN {X 0,Y 537.669,Z 205.255,A -85,B 0,C 180,E1 -3970.926,E2 -3970.926} C_VEL
LIN {X 0,Y 537.751,Z 196.991,A -85,B 0,C 180,E1 -3973.606,E2 -3973.606} C_VEL
LIN {X 0,Y 537.855,Z 188.774,A -85,B 0,C 180,E1 -3976.316,E2 -3976.316} C_VEL
LIN {X 0,Y 537.957,Z 180.464,A -85,B 0,C 180,E1 -3979.063,E2 -3979.063} C_VEL
LIN {X 0,Y 538.033,Z 171.764,A -85,B 0,C 180,E1 -3981.961,E2 -3981.961} C_VEL
LIN {X 0,Y 538.189,Z 163.657,A -85,B 0,C 180,E1 -3984.701,E2 -3984.701} C_VEL
LIN {X 0,Y 538.329,Z 155.703,A -85,B 0,C 180,E1 -3987.406,E2 -3987.406} C_VEL
LIN {X 0,Y 538.475,Z 148.999,A -85,B 0,C 180,E1 -3989.733,E2 -3989.733} C_VEL
LIN {X 0,Y 538.079,Z 145.464,A -85,B 0,C 180,E1 -3991.059,E2 -3991.059} C_VEL
LIN {X 0,Y 538.016,Z 145.47,A -85,B 0,C 180,E1 -3994.174,E2 -3994.174} C_VEL
LIN {X 0,Y 538.01,Z 145.472,A -85,B 0,C 180,E1 -3997.17,E2 -3997.17} C_VEL
LIN {X 0,Y 538.028,Z 145.468,A -85,B 0,C 180,E1 -3999.797,E2 -3999.797} C_VEL
LIN {X 0,Y 538.024,Z 145.469,A -85,B 0,C 180,E1 -4002.786,E2 -4002.786} C_VEL
LIN {X 0,Y 538.035,Z 145.469,A -85,B 0,C 180,E1 -4005.925,E2 -4005.925} C_VEL
LIN {X 0,Y 538.054,Z 145.466,A -85,B 0,C 180,E1 -4009.252,E2 -4009.252} C_VEL
LIN {X 0,Y 537.996,Z 145.473,A -85,B 0,C 180,E1 -4012.122,E2 -4012.122} C_VEL
LIN {X 0,Y 538.005,Z 145.471,A -85,B 0,C 180,E1 -4014.915,E2 -4014.915} C_VEL
LIN {X 0,Y 538.023,Z 145.471,A -85,B 0,C 180,E1 -4017.617,E2 -4017.617} C_VEL
LIN {X 0,Y 538.026,Z 145.475,A -85,B 0,C 180,E1 -4020.669,E2 -4020.669} C_VEL
LIN {X 0,Y 538.067,Z 145.633,A -85,B 0,C 180,E1 -4021.099,E2 -4021.099} C_VEL
LIN {X 0,Y 539.464,Z 152.542,A -85,B 0,C 180,E1 -4022.872,E2 -4022.872} C_VEL
LIN {X 0,Y 539.578,Z 157.348,A -85,B 0,C 180,E1 -4023.991,E2 -4023.991} C_VEL
LIN {X 0,Y 538.964,Z 171.15,A -85,B 0,C 180,E1 -4026.97,E2 -4026.97} C_VEL
LIN {X 0,Y 538.596,Z 185.913,A -85,B 0,C 180,E1 -4029.97,E2 -4029.97} C_VEL
LIN {X 0,Y 538.309,Z 201.161,A -85,B 0,C 180,E1 -4032.916,E2 -4032.916} C_VEL
LIN {X 0,Y 538.099,Z 217.399,A -85,B 0,C 180,E1 -4036.017,E2 -4036.017} C_VEL
LIN {X 0,Y 537.985,Z 220.924,A -85,B 0,C 180,E1 -4036.687,E2 -4036.687} C_VEL
LIN {X 0,Y 539.158,Z 230.382,A -85,B 0,C 180,E1 -4036.885,E2 -4036.885} C_VEL
LIN {X 0,Y 539.03,Z 243.198,A -85,B 0,C 180,E1 -4037.241,E2 -4037.241} C_VEL
LIN {X 0,Y 538.81,Z 255.013,A -85,B 0,C 180,E1 -4037.714,E2 -4037.714} C_VEL
LIN {X 0,Y 538.585,Z 266.105,A -85,B 0,C 180,E1 -4038.297,E2 -4038.297} C_VEL
LIN {X 0,Y 538.395,Z 277.917,A -85,B 0,C 180,E1 -4039.088,E2 -4039.088} C_VEL
LIN {X 0,Y 538.209,Z 287.013,A -85,B 0,C 180,E1 -4039.846,E2 -4039.846} C_VEL
LIN {X 0,Y 538.01,Z 296.326,A -85,B 0,C 180,E1 -4040.791,E2 -4040.791} C_VEL
LIN {X 0,Y 537.852,Z 305.372,A -85,B 0,C 180,E1 -4041.924,E2 -4041.924} C_VEL
LIN {X 0,Y 537.709,Z 312.644,A -85,B 0,C 180,E1 -4043.055,E2 -4043.055} C_VEL
LIN {X 0,Y 537.677,Z 319.261,A -85,B 0,C 180,E1 -4044.373,E2 -4044.373} C_VEL
LIN {X 0,Y 537.556,Z 323.626,A -85,B 0,C 180,E1 -4045.5,E2 -4045.5} C_VEL
LIN {X 0,Y 537.591,Z 325.936,A -85,B 0,C 180,E1 -4046.251,E2 -4046.251} C_VEL
LIN {X 0,Y 537.551,Z 327.797,A -85,B 0,C 180,E1 -4047.001,E2 -4047.001} C_VEL
LIN {X 0,Y 537.49,Z 329.189,A -85,B 0,C 180,E1 -4047.751,E2 -4047.751} C_VEL
LIN {X 0,Y 537.442,Z 330.784,A -85,B 0,C 180,E1 -4049.25,E2 -4049.25} C_VEL
LIN {X 0,Y 537.442,Z 331,A -85,B 0,C 180,E1 -4049.999,E2 -4049.999} C_VEL
LIN {X 0,Y 537.451,Z 330.184,A -85,B 0,C 180,E1 -4051.497,E2 -4051.497} C_VEL
LIN {X 0,Y 537.49,Z 329.195,A -85,B 0,C 180,E1 -4052.247,E2 -4052.247} C_VEL
LIN {X 0,Y 537.551,Z 327.806,A -85,B 0,C 180,E1 -4052.997,E2 -4052.997} C_VEL
LIN {X 0,Y 537.603,Z 324.871,A -85,B 0,C 180,E1 -4054.122,E2 -4054.122} C_VEL
LIN {X 0,Y 537.587,Z 320.874,A -85,B 0,C 180,E1 -4055.249,E2 -4055.249} C_VEL
LIN {X 0,Y 537.638,Z 315.986,A -85,B 0,C 180,E1 -4056.326,E2 -4056.326} C_VEL
LIN {X 0,Y 537.753,Z 309.242,A -85,B 0,C 180,E1 -4057.508,E2 -4057.508} C_VEL
LIN {X 0,Y 537.928,Z 301.148,A -85,B 0,C 180,E1 -4058.64,E2 -4058.64} C_VEL
LIN {X 0,Y 538.088,Z 292.886,A -85,B 0,C 180,E1 -4059.585,E2 -4059.585} C_VEL
LIN {X 0,Y 538.335,Z 282.796,A -85,B 0,C 180,E1 -4060.53,E2 -4060.53} C_VEL
LIN {X 0,Y 538.504,Z 272.779,A -85,B 0,C 180,E1 -4061.288,E2 -4061.288} C_VEL
LIN {X 0,Y 538.666,Z 261.783,A -85,B 0,C 180,E1 -4061.957,E2 -4061.957} C_VEL
LIN {X 0,Y 538.918,Z 248.701,A -85,B 0,C 180,E1 -4062.568,E2 -4062.568} C_VEL
LIN {X 0,Y 539.083,Z 235.77,A -85,B 0,C 180,E1 -4062.995,E2 -4062.995} C_VEL
LIN {X 0,Y 539.028,Z 228.125,A -85,B 0,C 180,E1 -4063.176,E2 -4063.176} C_VEL
LIN {X 0,Y 537.998,Z 220.963,A -85,B 0,C 180,E1 -4063.334,E2 -4063.334} C_VEL
LIN {X 0,Y 538.236,Z 205.264,A -85,B 0,C 180,E1 -4066.303,E2 -4066.303} C_VEL
LIN {X 0,Y 538.454,Z 190.947,A -85,B 0,C 180,E1 -4069.043,E2 -4069.043} C_VEL
LIN {X 0,Y 538.919,Z 175.183,A -85,B 0,C 180,E1 -4072.22,E2 -4072.22} C_VEL
LIN {X 0,Y 539.301,Z 160.35,A -85,B 0,C 180,E1 -4075.262,E2 -4075.262} C_VEL
LIN {X 0,Y 539.403,Z 153.295,A -85,B 0,C 180,E1 -4076.71,E2 -4076.71} C_VEL
LIN {X 0,Y 538.086,Z 145.708,A -85,B 0,C 180,E1 -4078.417,E2 -4078.417} C_VEL
LIN {X 0,Y 538.041,Z 145.468,A -85,B 0,C 180,E1 -4078.473,E2 -4078.473} C_VEL
LIN {X 0,Y 538.003,Z 145.468,A -85,B 0,C 180,E1 -4081.5,E2 -4081.5} C_VEL
LIN {X 0,Y 538.023,Z 145.471,A -85,B 0,C 180,E1 -4084.171,E2 -4084.171} C_VEL
LIN {X 0,Y 538.001,Z 145.471,A -85,B 0,C 180,E1 -4087.169,E2 -4087.169} C_VEL
LIN {X 0,Y 538.014,Z 145.466,A -85,B 0,C 180,E1 -4089.796,E2 -4089.796} C_VEL
LIN {X 0,Y 537.99,Z 145.471,A -85,B 0,C 180,E1 -4092.787,E2 -4092.787} C_VEL
LIN {X 0,Y 538.023,Z 145.465,A -85,B 0,C 180,E1 -4095.139,E2 -4095.139} C_VEL
LIN {X 0,Y 538.032,Z 145.464,A -85,B 0,C 180,E1 -4098.227,E2 -4098.227} C_VEL
LIN {X 0,Y 538.049,Z 145.463,A -85,B 0,C 180,E1 -4100.41,E2 -4100.41} C_VEL
LIN {X 0,Y 538.006,Z 145.467,A -85,B 0,C 180,E1 -4103.065,E2 -4103.065} C_VEL
LIN {X 0,Y 538.005,Z 145.471,A -85,B 0,C 180,E1 -4105.826,E2 -4105.826} C_VEL
LIN {X 0,Y 538.013,Z 145.466,A -85,B 0,C 180,E1 -4108.499,E2 -4108.499} C_VEL
LIN {X 0,Y 538.047,Z 145.467,A -85,B 0,C 180,E1 -4111.099,E2 -4111.099} C_VEL
LIN {X 0,Y 538.038,Z 145.463,A -85,B 0,C 180,E1 -4113.633,E2 -4113.633} C_VEL
LIN {X 0,Y 537.992,Z 145.472,A -85,B 0,C 180,E1 -4116.121,E2 -4116.121} C_VEL
LIN {X 0,Y 538.026,Z 145.47,A -85,B 0,C 180,E1 -4119.348,E2 -4119.348} C_VEL
LIN {X 0,Y 538.058,Z 145.465,A -85,B 0,C 180,E1 -4122.517,E2 -4122.517} C_VEL
LIN {X 0,Y 538.051,Z 145.463,A -85,B 0,C 180,E1 -4125.63,E2 -4125.63} C_VEL
LIN {X 0,Y 538.059,Z 145.46,A -85,B 0,C 180,E1 -4128.701,E2 -4128.701} C_VEL
LIN {X 0,Y 538.066,Z 145.459,A -85,B 0,C 180,E1 -4131.739,E2 -4131.739} C_VEL
LIN {X 0,Y 538.171,Z 145.449,A -85,B 0,C 180,E1 -4134.755,E2 -4134.755} C_VEL
LIN {X 0,Y 538.155,Z 145.453,A -85,B 0,C 180,E1 -4137.755,E2 -4137.755} C_VEL
LIN {X 0,Y 538.167,Z 145.448,A -85,B 0,C 180,E1 -4140.748,E2 -4140.748} C_VEL
LIN {X 0,Y 538.118,Z 145.457,A -85,B 0,C 180,E1 -4142.995,E2 -4142.995} C_VEL
LIN {X 0,Y 538.108,Z 145.458,A -85,B 0,C 180,E1 -4145.997,E2 -4145.997} C_VEL
LIN {X 0,Y 538.066,Z 145.46,A -85,B 0,C 180,E1 -4149.018,E2 -4149.018} C_VEL
LIN {X 0,Y 538.068,Z 145.459,A -85,B 0,C 180,E1 -4152.063,E2 -4152.063} C_VEL
LIN {X 0,Y 538.029,Z 145.464,A -85,B 0,C 180,E1 -4155.144,E2 -4155.144} C_VEL
LIN {X 0,Y 538.021,Z 145.468,A -85,B 0,C 180,E1 -4158.271,E2 -4158.271} C_VEL
LIN {X 0,Y 538.03,Z 145.464,A -85,B 0,C 180,E1 -4160.652,E2 -4160.652} C_VEL
LIN {X 0,Y 538.028,Z 145.464,A -85,B 0,C 180,E1 -4163.887,E2 -4163.887} C_VEL
LIN {X 0,Y 538.02,Z 145.47,A -85,B 0,C 180,E1 -4166.368,E2 -4166.368} C_VEL
LIN {X 0,Y 538.016,Z 145.465,A -85,B 0,C 180,E1 -4168.934,E2 -4168.934} C_VEL
LIN {X 0,Y 538.015,Z 145.467,A -85,B 0,C 180,E1 -4171.891,E2 -4171.891} C_VEL
LIN {X 0,Y 538.024,Z 145.47,A -85,B 0,C 180,E1 -4174.623,E2 -4174.623} C_VEL
LIN {X 0,Y 537.996,Z 145.468,A -85,B 0,C 180,E1 -4177.172,E2 -4177.172} C_VEL
LIN {X 0,Y 538.005,Z 145.467,A -85,B 0,C 180,E1 -4180.283,E2 -4180.283} C_VEL
LIN {X 0,Y 537.358,Z 145.548,A -85,B 0,C 180,E1 -4180.908,E2 -4180.908} C_VEL
LIN {X 0,Y 534.51,Z 145.904,A -85,B 0,C 180,E1 -4181.923,E2 -4181.923} C_VEL
LIN {X 0,Y 532.087,Z 146.208,A -85,B 0,C 180,E1 -4182.74,E2 -4182.74} C_VEL
LIN {X 0,Y 531.04,Z 146.338,A -85,B 0,C 180,E1 -4183.371,E2 -4183.371} C_VEL
LIN {X 0,Y 530.952,Z 146.347,A -85,B 0,C 180,E1 -4183.585,E2 -4183.585} C_VEL
LIN {X 0,Y 530.958,Z 146.349,A -85,B 0,C 180,E1 -4186.507,E2 -4186.507} C_VEL
LIN {X 0,Y 530.981,Z 146.342,A -85,B 0,C 180,E1 -4188.977,E2 -4188.977} C_VEL
LIN {X 0,Y 530.945,Z 146.352,A -85,B 0,C 180,E1 -4191.53,E2 -4191.53} C_VEL
LIN {X 0,Y 530.943,Z 146.347,A -85,B 0,C 180,E1 -4194.381,E2 -4194.381} C_VEL
LIN {X 0,Y 530.966,Z 146.344,A -85,B 0,C 180,E1 -4197.135,E2 -4197.135} C_VEL
LIN {X 0,Y 530.982,Z 146.347,A -85,B 0,C 180,E1 -4199.806,E2 -4199.806} C_VEL
LIN {X 0,Y 531.011,Z 146.338,A -85,B 0,C 180,E1 -4202.468,E2 -4202.468} C_VEL
LIN {X 0,Y 530.95,Z 146.352,A -85,B 0,C 180,E1 -4204.941,E2 -4204.941} C_VEL
LIN {X 0,Y 530.972,Z 146.344,A -85,B 0,C 180,E1 -4207.9,E2 -4207.9} C_VEL
LIN {X 0,Y 530.993,Z 146.341,A -85,B 0,C 180,E1 -4210.679,E2 -4210.679} C_VEL
LIN {X 0,Y 530.984,Z 146.345,A -85,B 0,C 180,E1 -4213.072,E2 -4213.072} C_VEL
LIN {X 0,Y 531.011,Z 146.34,A -85,B 0,C 180,E1 -4215.437,E2 -4215.437} C_VEL
LIN {X 0,Y 531.034,Z 146.339,A -85,B 0,C 180,E1 -4218.551,E2 -4218.551} C_VEL
LIN {X 0,Y 531.051,Z 146.337,A -85,B 0,C 180,E1 -4221.631,E2 -4221.631} C_VEL
LIN {X 0,Y 531.121,Z 146.327,A -85,B 0,C 180,E1 -4224.687,E2 -4224.687} C_VEL
LIN {X 0,Y 531.14,Z 146.322,A -85,B 0,C 180,E1 -4227.726,E2 -4227.726} C_VEL
LIN {X 0,Y 531.13,Z 146.328,A -85,B 0,C 180,E1 -4230.001,E2 -4230.001} C_VEL
LIN {X 0,Y 531.098,Z 146.328,A -85,B 0,C 180,E1 -4233.035,E2 -4233.035} C_VEL
LIN {X 0,Y 531.087,Z 146.329,A -85,B 0,C 180,E1 -4236.078,E2 -4236.078} C_VEL
LIN {X 0,Y 531.055,Z 146.338,A -85,B 0,C 180,E1 -4238.372,E2 -4238.372} C_VEL
LIN {X 0,Y 531.053,Z 146.337,A -85,B 0,C 180,E1 -4241.672,E2 -4241.672} C_VEL
LIN {X 0,Y 531.022,Z 146.339,A -85,B 0,C 180,E1 -4244.951,E2 -4244.951} C_VEL
LIN {X 0,Y 530.986,Z 146.341,A -85,B 0,C 180,E1 -4247.724,E2 -4247.724} C_VEL
LIN {X 0,Y 531.03,Z 146.341,A -85,B 0,C 180,E1 -4250.128,E2 -4250.128} C_VEL
LIN {X 0,Y 530.945,Z 146.347,A -85,B 0,C 180,E1 -4252.574,E2 -4252.574} C_VEL
LIN {X 0,Y 530.95,Z 146.349,A -85,B 0,C 180,E1 -4255.061,E2 -4255.061} C_VEL
LIN {X 0,Y 530.962,Z 146.344,A -85,B 0,C 180,E1 -4257.599,E2 -4257.599} C_VEL
LIN {X 0,Y 530.967,Z 146.347,A -85,B 0,C 180,E1 -4260.643,E2 -4260.643} C_VEL
LIN {X 0,Y 530.967,Z 146.348,A -85,B 0,C 180,E1 -4263.5,E2 -4263.5} C_VEL
LIN {X 0,Y 530.94,Z 146.347,A -85,B 0,C 180,E1 -4266.152,E2 -4266.152} C_VEL
LIN {X 0,Y 530.946,Z 146.351,A -85,B 0,C 180,E1 -4268.651,E2 -4268.651} C_VEL
LIN {X 0,Y 530.968,Z 146.344,A -85,B 0,C 180,E1 -4271.439,E2 -4271.439} C_VEL
LIN {X 0,Y 530.978,Z 146.343,A -85,B 0,C 180,E1 -4274.549,E2 -4274.549} C_VEL
LIN {X 0,Y 530.986,Z 146.341,A -85,B 0,C 180,E1 -4277.835,E2 -4277.835} C_VEL
LIN {X 0,Y 530.972,Z 146.347,A -85,B 0,C 180,E1 -4280.555,E2 -4280.555} C_VEL
LIN {X 0,Y 530.939,Z 146.353,A -85,B 0,C 180,E1 -4283.849,E2 -4283.849} C_VEL
LIN {X 0,Y 530.967,Z 146.344,A -85,B 0,C 180,E1 -4286.501,E2 -4286.501} C_VEL
LIN {X 0,Y 531.03,Z 146.37,A -85,B 0,C 180,E1 -4289.043,E2 -4289.043} C_VEL
LIN {X 0,Y 531.397,Z 151.219,A -85,B 0,C 180,E1 -4290.797,E2 -4290.797} C_VEL
LIN {X 0,Y 531.24,Z 159.471,A -85,B 0,C 180,E1 -4293.693,E2 -4293.693} C_VEL
LIN {X 0,Y 531.039,Z 167.937,A -85,B 0,C 180,E1 -4296.607,E2 -4296.607} C_VEL
LIN {X 0,Y 530.968,Z 176.389,A -85,B 0,C 180,E1 -4299.466,E2 -4299.466} C_VEL
LIN {X 0,Y 530.842,Z 185.26,A -85,B 0,C 180,E1 -4302.409,E2 -4302.409} C_VEL
LIN {X 0,Y 530.722,Z 194.273,A -85,B 0,C 180,E1 -4305.428,E2 -4305.428} C_VEL
LIN {X 0,Y 530.618,Z 203.732,A -85,B 0,C 180,E1 -4308.56,E2 -4308.56} C_VEL
LIN {X 0,Y 530.532,Z 213.17,A -85,B 0,C 180,E1 -4311.621,E2 -4311.621} C_VEL
LIN {X 0,Y 530.507,Z 214.45,A -85,B 0,C 180,E1 -4312.028,E2 -4312.028} C_VEL
LIN {X 0,Y 531.15,Z 223.953,A -85,B 0,C 180,E1 -4312.397,E2 -4312.397} C_VEL
LIN {X 0,Y 530.997,Z 233.479,A -85,B 0,C 180,E1 -4312.901,E2 -4312.901} C_VEL
LIN {X 0,Y 530.869,Z 242.21,A -85,B 0,C 180,E1 -4313.53,E2 -4313.53} C_VEL
LIN {X 0,Y 530.709,Z 250.201,A -85,B 0,C 180,E1 -4314.3,E2 -4314.3} C_VEL
LIN {X 0,Y 530.72,Z 256.317,A -85,B 0,C 180,E1 -4315.062,E2 -4315.062} C_VEL
LIN {X 0,Y 530.62,Z 261.138,A -85,B 0,C 180,E1 -4315.823,E2 -4315.823} C_VEL
LIN {X 0,Y 530.584,Z 264.892,A -85,B 0,C 180,E1 -4316.583,E2 -4316.583} C_VEL
LIN {X 0,Y 530.431,Z 268.911,A -85,B 0,C 180,E1 -4317.722,E2 -4317.722} C_VEL
LIN {X 0,Y 530.383,Z 270.659,A -85,B 0,C 180,E1 -4318.481,E2 -4318.481} C_VEL
LIN {X 0,Y 530.373,Z 271.709,A -85,B 0,C 180,E1 -4319.241,E2 -4319.241} C_VEL
LIN {X 0,Y 530.372,Z 272.093,A -85,B 0,C 180,E1 -4320,E2 -4320} C_VEL
LIN {X 0,Y 530.374,Z 271.818,A -85,B 0,C 180,E1 -4320.759,E2 -4320.759} C_VEL
LIN {X 0,Y 530.385,Z 270.879,A -85,B 0,C 180,E1 -4321.519,E2 -4321.519} C_VEL
LIN {X 0,Y 530.476,Z 268.139,A -85,B 0,C 180,E1 -4322.658,E2 -4322.658} C_VEL
LIN {X 0,Y 530.583,Z 265.392,A -85,B 0,C 180,E1 -4323.417,E2 -4323.417} C_VEL
LIN {X 0,Y 530.618,Z 260.734,A -85,B 0,C 180,E1 -4324.368,E2 -4324.368} C_VEL
LIN {X 0,Y 530.692,Z 255.807,A -85,B 0,C 180,E1 -4325.129,E2 -4325.129} C_VEL
LIN {X 0,Y 530.695,Z 249.571,A -85,B 0,C 180,E1 -4325.891,E2 -4325.891} C_VEL
LIN {X 0,Y 530.881,Z 242.384,A -85,B 0,C 180,E1 -4326.575,E2 -4326.575} C_VEL
LIN {X 0,Y 531.006,Z 233.431,A -85,B 0,C 180,E1 -4327.223,E2 -4327.223} C_VEL
LIN {X 0,Y 531.217,Z 223.479,A -85,B 0,C 180,E1 -4327.746,E2 -4327.746} C_VEL
LIN {X 0,Y 530.662,Z 215.772,A -85,B 0,C 180,E1 -4328.041,E2 -4328.041} C_VEL
LIN {X 0,Y 530.548,Z 214.666,A -85,B 0,C 180,E1 -4328.091,E2 -4328.091} C_VEL
LIN {X 0,Y 530.615,Z 205.488,A -85,B 0,C 180,E1 -4331.068,E2 -4331.068} C_VEL
LIN {X 0,Y 530.705,Z 197.21,A -85,B 0,C 180,E1 -4333.79,E2 -4333.79} C_VEL
LIN {X 0,Y 530.807,Z 188.936,A -85,B 0,C 180,E1 -4336.539,E2 -4336.539} C_VEL
LIN {X 0,Y 530.919,Z 180.562,A -85,B 0,C 180,E1 -4339.326,E2 -4339.326} C_VEL
LIN {X 0,Y 531.016,Z 172.346,A -85,B 0,C 180,E1 -4342.111,E2 -4342.111} C_VEL
LIN {X 0,Y 531.147,Z 163.735,A -85,B 0,C 180,E1 -4345.051,E2 -4345.051} C_VEL
LIN {X 0,Y 531.341,Z 156.424,A -85,B 0,C 180,E1 -4347.599,E2 -4347.599} C_VEL
LIN {X 0,Y 531.508,Z 150.444,A -85,B 0,C 180,E1 -4349.726,E2 -4349.726} C_VEL
LIN {X 0,Y 531,Z 146.347,A -85,B 0,C 180,E1 -4351.298,E2 -4351.298} C_VEL
LIN {X 0,Y 530.961,Z 146.35,A -85,B 0,C 180,E1 -4353.775,E2 -4353.775} C_VEL
LIN {X 0,Y 530.961,Z 146.349,A -85,B 0,C 180,E1 -4356.558,E2 -4356.558} C_VEL
LIN {X 0,Y 530.991,Z 146.346,A -85,B 0,C 180,E1 -4359.443,E2 -4359.443} C_VEL
LIN {X 0,Y 530.983,Z 146.348,A -85,B 0,C 180,E1 -4362.456,E2 -4362.456} C_VEL
LIN {X 0,Y 530.988,Z 146.346,A -85,B 0,C 180,E1 -4365.621,E2 -4365.621} C_VEL
LIN {X 0,Y 531,Z 146.343,A -85,B 0,C 180,E1 -4368.564,E2 -4368.564} C_VEL
LIN {X 0,Y 530.961,Z 146.349,A -85,B 0,C 180,E1 -4371.529,E2 -4371.529} C_VEL
LIN {X 0,Y 530.961,Z 146.35,A -85,B 0,C 180,E1 -4374.379,E2 -4374.379} C_VEL
LIN {X 0,Y 530.972,Z 146.349,A -85,B 0,C 180,E1 -4377.133,E2 -4377.133} C_VEL
LIN {X 0,Y 530.975,Z 146.353,A -85,B 0,C 180,E1 -4379.802,E2 -4379.802} C_VEL
LIN {X 0,Y 531.002,Z 146.478,A -85,B 0,C 180,E1 -4380.745,E2 -4380.745} C_VEL
LIN {X 0,Y 532.654,Z 154.671,A -85,B 0,C 180,E1 -4382.921,E2 -4382.921} C_VEL
LIN {X 0,Y 532.589,Z 160.087,A -85,B 0,C 180,E1 -4384.184,E2 -4384.184} C_VEL
LIN {X 0,Y 532.063,Z 171.349,A -85,B 0,C 180,E1 -4386.654,E2 -4386.654} C_VEL
LIN {X 0,Y 531.697,Z 182.902,A -85,B 0,C 180,E1 -4389.09,E2 -4389.09} C_VEL
LIN {X 0,Y 531.362,Z 198.936,A -85,B 0,C 180,E1 -4392.289,E2 -4392.289} C_VEL
LIN {X 0,Y 531.001,Z 215.102,A -85,B 0,C 180,E1 -4395.434,E2 -4395.434} C_VEL
LIN {X 0,Y 530.937,Z 220.999,A -85,B 0,C 180,E1 -4396.556,E2 -4396.556} C_VEL
LIN {X 0,Y 532.179,Z 230.596,A -85,B 0,C 180,E1 -4396.758,E2 -4396.758} C_VEL
LIN {X 0,Y 532.023,Z 243.238,A -85,B 0,C 180,E1 -4397.118,E2 -4397.118} C_VEL
LIN {X 0,Y 531.765,Z 255.993,A -85,B 0,C 180,E1 -4397.646,E2 -4397.646} C_VEL
LIN {X 0,Y 531.54,Z 266.683,A -85,B 0,C 180,E1 -4398.227,E2 -4398.227} C_VEL
LIN {X 0,Y 531.389,Z 277.169,A -85,B 0,C 180,E1 -4398.943,E2 -4398.943} C_VEL
LIN {X 0,Y 531.136,Z 287.377,A -85,B 0,C 180,E1 -4399.805,E2 -4399.805} C_VEL
LIN {X 0,Y 530.93,Z 297.397,A -85,B 0,C 180,E1 -4400.859,E2 -4400.859} C_VEL
LIN {X 0,Y 530.756,Z 306.201,A -85,B 0,C 180,E1 -4402.007,E2 -4402.007} C_VEL
LIN {X 0,Y 530.592,Z 313.201,A -85,B 0,C 180,E1 -4403.152,E2 -4403.152} C_VEL
LIN {X 0,Y 530.591,Z 318.81,A -85,B 0,C 180,E1 -4404.298,E2 -4404.298} C_VEL
LIN {X 0,Y 530.455,Z 323.196,A -85,B 0,C 180,E1 -4405.439,E2 -4405.439} C_VEL
LIN {X 0,Y 530.516,Z 325.521,A -85,B 0,C 180,E1 -4406.201,E2 -4406.201} C_VEL
LIN {X 0,Y 530.457,Z 327.404,A -85,B 0,C 180,E1 -4406.961,E2 -4406.961} C_VEL
LIN {X 0,Y 530.411,Z 328.813,A -85,B 0,C 180,E1 -4407.721,E2 -4407.721} C_VEL
LIN {X 0,Y 530.35,Z 330.432,A -85,B 0,C 180,E1 -4409.24,E2 -4409.24} C_VEL
LIN {X 0,Y 530.351,Z 330.653,A -85,B 0,C 180,E1 -4409.999,E2 -4409.999} C_VEL
LIN {X 0,Y 530.35,Z 330.437,A -85,B 0,C 180,E1 -4410.758,E2 -4410.758} C_VEL
LIN {X 0,Y 530.411,Z 328.83,A -85,B 0,C 180,E1 -4412.277,E2 -4412.277} C_VEL
LIN {X 0,Y 530.457,Z 327.426,A -85,B 0,C 180,E1 -4413.037,E2 -4413.037} C_VEL
LIN {X 0,Y 530.522,Z 324.472,A -85,B 0,C 180,E1 -4414.177,E2 -4414.177} C_VEL
LIN {X 0,Y 530.524,Z 320.463,A -85,B 0,C 180,E1 -4415.319,E2 -4415.319} C_VEL
LIN {X 0,Y 530.592,Z 314.705,A -85,B 0,C 180,E1 -4416.575,E2 -4416.575} C_VEL
LIN {X 0,Y 530.718,Z 307.536,A -85,B 0,C 180,E1 -4417.8,E2 -4417.8} C_VEL
LIN {X 0,Y 530.913,Z 299.153,A -85,B 0,C 180,E1 -4418.947,E2 -4418.947} C_VEL
LIN {X 0,Y 531.069,Z 290.501,A -85,B 0,C 180,E1 -4419.905,E2 -4419.905} C_VEL
LIN {X 0,Y 531.345,Z 279.824,A -85,B 0,C 180,E1 -4420.863,E2 -4420.863} C_VEL
LIN {X 0,Y 531.576,Z 268.846,A -85,B 0,C 180,E1 -4421.655,E2 -4421.655} C_VEL
LIN {X 0,Y 531.781,Z 257.408,A -85,B 0,C 180,E1 -4422.303,E2 -4422.303} C_VEL
LIN {X 0,Y 532.016,Z 245.102,A -85,B 0,C 180,E1 -4422.831,E2 -4422.831} C_VEL
LIN {X 0,Y 532.173,Z 232.548,A -85,B 0,C 180,E1 -4423.215,E2 -4423.215} C_VEL
LIN {X 0,Y 531.777,Z 226.961,A -85,B 0,C 180,E1 -4423.347,E2 -4423.347} C_VEL
LIN {X 0,Y 530.951,Z 220.876,A -85,B 0,C 180,E1 -4423.49,E2 -4423.49} C_VEL
LIN {X 0,Y 531.192,Z 205.138,A -85,B 0,C 180,E1 -4426.525,E2 -4426.525} C_VEL
LIN {X 0,Y 531.411,Z 192.866,A -85,B 0,C 180,E1 -4428.904,E2 -4428.904} C_VEL
LIN {X 0,Y 531.751,Z 181.04,A -85,B 0,C 180,E1 -4431.311,E2 -4431.311} C_VEL
LIN {X 0,Y 532.26,Z 166.397,A -85,B 0,C 180,E1 -4434.344,E2 -4434.344} C_VEL
LIN {X 0,Y 532.54,Z 155.362,A -85,B 0,C 180,E1 -4436.659,E2 -4436.659} C_VEL
LIN {X 0,Y 531.578,Z 149.345,A -85,B 0,C 180,E1 -4438.013,E2 -4438.013} C_VEL
LIN {X 0,Y 530.974,Z 146.349,A -85,B 0,C 180,E1 -4438.763,E2 -4438.763} C_VEL
LIN {X 0,Y 530.966,Z 146.347,A -85,B 0,C 180,E1 -4441.966,E2 -4441.966} C_VEL
LIN {X 0,Y 530.984,Z 146.342,A -85,B 0,C 180,E1 -4444.853,E2 -4444.853} C_VEL
LIN {X 0,Y 530.96,Z 146.349,A -85,B 0,C 180,E1 -4447.506,E2 -4447.506} C_VEL
LIN {X 0,Y 530.956,Z 146.347,A -85,B 0,C 180,E1 -4450.433,E2 -4450.433} C_VEL
LIN {X 0,Y 530.934,Z 146.347,A -85,B 0,C 180,E1 -4453.278,E2 -4453.278} C_VEL
LIN {X 0,Y 530.979,Z 146.346,A -85,B 0,C 180,E1 -4455.619,E2 -4455.619} C_VEL
LIN {X 0,Y 530.998,Z 146.34,A -85,B 0,C 180,E1 -4458.565,E2 -4458.565} C_VEL
LIN {X 0,Y 530.957,Z 146.346,A -85,B 0,C 180,E1 -4461.345,E2 -4461.345} C_VEL
LIN {X 0,Y 530.936,Z 146.351,A -85,B 0,C 180,E1 -4464.378,E2 -4464.378} C_VEL
LIN {X 0,Y 530.96,Z 146.346,A -85,B 0,C 180,E1 -4467.133,E2 -4467.133} C_VEL
LIN {X 0,Y 530.974,Z 146.344,A -85,B 0,C 180,E1 -4469.803,E2 -4469.803} C_VEL
LIN {X 0,Y 531.005,Z 146.344,A -85,B 0,C 180,E1 -4472.465,E2 -4472.465} C_VEL
LIN {X 0,Y 530.983,Z 146.342,A -85,B 0,C 180,E1 -4474.941,E2 -4474.941} C_VEL
LIN {X 0,Y 530.957,Z 146.345,A -85,B 0,C 180,E1 -4478.246,E2 -4478.246} C_VEL
LIN {X 0,Y 530.984,Z 146.344,A -85,B 0,C 180,E1 -4480.677,E2 -4480.677} C_VEL
LIN {X 0,Y 530.981,Z 146.344,A -85,B 0,C 180,E1 -4483.071,E2 -4483.071} C_VEL
LIN {X 0,Y 531.006,Z 146.339,A -85,B 0,C 180,E1 -4485.435,E2 -4485.435} C_VEL
LIN {X 0,Y 531.031,Z 146.335,A -85,B 0,C 180,E1 -4488.55,E2 -4488.55} C_VEL
LIN {X 0,Y 531.035,Z 146.336,A -85,B 0,C 180,E1 -4491.629,E2 -4491.629} C_VEL
LIN {X 0,Y 531.127,Z 146.328,A -85,B 0,C 180,E1 -4494.685,E2 -4494.685} C_VEL
LIN {X 0,Y 531.127,Z 146.329,A -85,B 0,C 180,E1 -4497.725,E2 -4497.725} C_VEL
LIN {X 0,Y 531.137,Z 146.324,A -85,B 0,C 180,E1 -4500.758,E2 -4500.758} C_VEL
LIN {X 0,Y 531.084,Z 146.332,A -85,B 0,C 180,E1 -4503.034,E2 -4503.034} C_VEL
LIN {X 0,Y 531.068,Z 146.335,A -85,B 0,C 180,E1 -4506.077,E2 -4506.077} C_VEL
LIN {X 0,Y 531.025,Z 146.339,A -85,B 0,C 180,E1 -4509.138,E2 -4509.138} C_VEL
LIN {X 0,Y 531.025,Z 146.336,A -85,B 0,C 180,E1 -4512.225,E2 -4512.225} C_VEL
LIN {X 0,Y 530.98,Z 146.341,A -85,B 0,C 180,E1 -4515.35,E2 -4515.35} C_VEL
LIN {X 0,Y 531.002,Z 146.342,A -85,B 0,C 180,E1 -4517.723,E2 -4517.723} C_VEL
LIN {X 0,Y 530.992,Z 146.343,A -85,B 0,C 180,E1 -4520.938,E2 -4520.938} C_VEL
LIN {X 0,Y 530.994,Z 146.341,A -85,B 0,C 180,E1 -4524.046,E2 -4524.046} C_VEL
LIN {X 0,Y 530.971,Z 146.344,A -85,B 0,C 180,E1 -4526.745,E2 -4526.745} C_VEL
LIN {X 0,Y 530.974,Z 146.344,A -85,B 0,C 180,E1 -4529.323,E2 -4529.323} C_VEL
LIN {X 0,Y 530.968,Z 146.344,A -85,B 0,C 180,E1 -4532.104,E2 -4532.104} C_VEL
LIN {X 0,Y 530.98,Z 146.346,A -85,B 0,C 180,E1 -4534.856,E2 -4534.856} C_VEL
LIN {X 0,Y 530.954,Z 146.346,A -85,B 0,C 180,E1 -4537.509,E2 -4537.509} C_VEL
LIN {X 0,Y 530.969,Z 146.342,A -85,B 0,C 180,E1 -4540.434,E2 -4540.434} C_VEL
LIN {X 0,Y 530.956,Z 146.347,A -85,B 0,C 180,E1 -4543.496,E2 -4543.496} C_VEL
LIN {X 0,Y 530.952,Z 146.347,A -85,B 0,C 180,E1 -4543.585,E2 -4543.585} C_VEL
LIN {X 0,Y 530.281,Z 146.431,A -85,B 0,C 180,E1 -4544.219,E2 -4544.219} C_VEL
LIN {X 0,Y 527.434,Z 146.786,A -85,B 0,C 180,E1 -4545.247,E2 -4545.247} C_VEL
LIN {X 0,Y 525.031,Z 147.088,A -85,B 0,C 180,E1 -4546.076,E2 -4546.076} C_VEL
LIN {X 0,Y 523.998,Z 147.216,A -85,B 0,C 180,E1 -4546.716,E2 -4546.716} C_VEL
LIN {X 0,Y 523.914,Z 147.224,A -85,B 0,C 180,E1 -4546.932,E2 -4546.932} C_VEL
LIN {X 0,Y 523.94,Z 147.223,A -85,B 0,C 180,E1 -4549.922,E2 -4549.922} C_VEL
LIN {X 0,Y 523.896,Z 147.226,A -85,B 0,C 180,E1 -4552.869,E2 -4552.869} C_VEL
LIN {X 0,Y 523.925,Z 147.221,A -85,B 0,C 180,E1 -4555.711,E2 -4555.711} C_VEL
LIN {X 0,Y 523.928,Z 147.225,A -85,B 0,C 180,E1 -4558.458,E2 -4558.458} C_VEL
LIN {X 0,Y 523.939,Z 147.221,A -85,B 0,C 180,E1 -4561.127,E2 -4561.127} C_VEL
LIN {X 0,Y 523.937,Z 147.219,A -85,B 0,C 180,E1 -4563.991,E2 -4563.991} C_VEL
LIN {X 0,Y 523.902,Z 147.224,A -85,B 0,C 180,E1 -4567.108,E2 -4567.108} C_VEL
LIN {X 0,Y 523.977,Z 147.218,A -85,B 0,C 180,E1 -4569.867,E2 -4569.867} C_VEL
LIN {X 0,Y 523.965,Z 147.217,A -85,B 0,C 180,E1 -4572.839,E2 -4572.839} C_VEL
LIN {X 0,Y 523.971,Z 147.218,A -85,B 0,C 180,E1 -4575.237,E2 -4575.237} C_VEL
LIN {X 0,Y 524.013,Z 147.216,A -85,B 0,C 180,E1 -4578.396,E2 -4578.396} C_VEL
LIN {X 0,Y 523.999,Z 147.215,A -85,B 0,C 180,E1 -4581.517,E2 -4581.517} C_VEL
LIN {X 0,Y 524.083,Z 147.203,A -85,B 0,C 180,E1 -4584.615,E2 -4584.615} C_VEL
LIN {X 0,Y 524.113,Z 147.198,A -85,B 0,C 180,E1 -4587.696,E2 -4587.696} C_VEL
LIN {X 0,Y 524.099,Z 147.204,A -85,B 0,C 180,E1 -4590.001,E2 -4590.001} C_VEL
LIN {X 0,Y 524.04,Z 147.208,A -85,B 0,C 180,E1 -4593.076,E2 -4593.076} C_VEL
LIN {X 0,Y 524.05,Z 147.206,A -85,B 0,C 180,E1 -4596.16,E2 -4596.16} C_VEL
LIN {X 0,Y 524.003,Z 147.216,A -85,B 0,C 180,E1 -4598.485,E2 -4598.485} C_VEL
LIN {X 0,Y 524.002,Z 147.216,A -85,B 0,C 180,E1 -4601.738,E2 -4601.738} C_VEL
LIN {X 0,Y 523.986,Z 147.216,A -85,B 0,C 180,E1 -4605.048,E2 -4605.048} C_VEL
LIN {X 0,Y 523.952,Z 147.218,A -85,B 0,C 180,E1 -4607.97,E2 -4607.97} C_VEL
LIN {X 0,Y 523.977,Z 147.219,A -85,B 0,C 180,E1 -4610.411,E2 -4610.411} C_VEL
LIN {X 0,Y 523.911,Z 147.223,A -85,B 0,C 180,E1 -4612.895,E2 -4612.895} C_VEL
LIN {X 0,Y 523.901,Z 147.228,A -85,B 0,C 180,E1 -4615.422,E2 -4615.422} C_VEL
LIN {X 0,Y 523.913,Z 147.222,A -85,B 0,C 180,E1 -4618.003,E2 -4618.003} C_VEL
LIN {X 0,Y 523.941,Z 147.22,A -85,B 0,C 180,E1 -4620.854,E2 -4620.854} C_VEL
LIN {X 0,Y 523.935,Z 147.224,A -85,B 0,C 180,E1 -4623.73,E2 -4623.73} C_VEL
LIN {X 0,Y 523.893,Z 147.225,A -85,B 0,C 180,E1 -4626.4,E2 -4626.4} C_VEL
LIN {X 0,Y 523.903,Z 147.225,A -85,B 0,C 180,E1 -4629.087,E2 -4629.087} C_VEL
LIN {X 0,Y 523.936,Z 147.225,A -85,B 0,C 180,E1 -4632.121,E2 -4632.121} C_VEL
LIN {X 0,Y 523.947,Z 147.223,A -85,B 0,C 180,E1 -4635.311,E2 -4635.311} C_VEL
LIN {X 0,Y 523.96,Z 147.222,A -85,B 0,C 180,E1 -4638.69,E2 -4638.69} C_VEL
LIN {X 0,Y 523.905,Z 147.225,A -85,B 0,C 180,E1 -4641.897,E2 -4641.897} C_VEL
LIN {X 0,Y 523.926,Z 147.221,A -85,B 0,C 180,E1 -4644.912,E2 -4644.912} C_VEL
LIN {X 0,Y 523.94,Z 147.222,A -85,B 0,C 180,E1 -4647.68,E2 -4647.68} C_VEL
LIN {X 0,Y 524.002,Z 147.223,A -85,B 0,C 180,E1 -4648.921,E2 -4648.921} C_VEL
LIN {X 0,Y 524.406,Z 151.774,A -85,B 0,C 180,E1 -4650.59,E2 -4650.59} C_VEL
LIN {X 0,Y 524.213,Z 160.664,A -85,B 0,C 180,E1 -4653.741,E2 -4653.741} C_VEL
LIN {X 0,Y 524.014,Z 169.146,A -85,B 0,C 180,E1 -4656.693,E2 -4656.693} C_VEL
LIN {X 0,Y 523.875,Z 178.52,A -85,B 0,C 180,E1 -4659.899,E2 -4659.899} C_VEL
LIN {X 0,Y 523.771,Z 187.259,A -85,B 0,C 180,E1 -4662.831,E2 -4662.831} C_VEL
LIN {X 0,Y 523.652,Z 195.522,A -85,B 0,C 180,E1 -4665.624,E2 -4665.624} C_VEL
LIN {X 0,Y 523.551,Z 204.109,A -85,B 0,C 180,E1 -4668.504,E2 -4668.504} C_VEL
LIN {X 0,Y 523.463,Z 213.315,A -85,B 0,C 180,E1 -4671.507,E2 -4671.507} C_VEL
LIN {X 0,Y 523.451,Z 214.519,A -85,B 0,C 180,E1 -4671.896,E2 -4671.896} C_VEL
LIN {X 0,Y 524.173,Z 223.454,A -85,B 0,C 180,E1 -4672.246,E2 -4672.246} C_VEL
LIN {X 0,Y 523.998,Z 233.484,A -85,B 0,C 180,E1 -4672.777,E2 -4672.777} C_VEL
LIN {X 0,Y 523.846,Z 241.929,A -85,B 0,C 180,E1 -4673.388,E2 -4673.388} C_VEL
LIN {X 0,Y 523.663,Z 248.818,A -85,B 0,C 180,E1 -4674.03,E2 -4674.03} C_VEL
LIN {X 0,Y 523.647,Z 255.278,A -85,B 0,C 180,E1 -4674.802,E2 -4674.802} C_VEL
LIN {X 0,Y 523.546,Z 261.495,A -85,B 0,C 180,E1 -4675.766,E2 -4675.766} C_VEL
LIN {X 0,Y 523.525,Z 265.254,A -85,B 0,C 180,E1 -4676.537,E2 -4676.537} C_VEL
LIN {X 0,Y 523.356,Z 269.289,A -85,B 0,C 180,E1 -4677.691,E2 -4677.691} C_VEL
LIN {X 0,Y 523.296,Z 271.043,A -85,B 0,C 180,E1 -4678.461,E2 -4678.461} C_VEL
LIN {X 0,Y 523.285,Z 272.1,A -85,B 0,C 180,E1 -4679.231,E2 -4679.231} C_VEL
LIN {X 0,Y 523.283,Z 272.489,A -85,B 0,C 180,E1 -4680,E2 -4680} C_VEL
LIN {X 0,Y 523.286,Z 272.217,A -85,B 0,C 180,E1 -4680.77,E2 -4680.77} C_VEL
LIN {X 0,Y 523.299,Z 271.28,A -85,B 0,C 180,E1 -4681.539,E2 -4681.539} C_VEL
LIN {X 0,Y 523.402,Z 268.549,A -85,B 0,C 180,E1 -4682.694,E2 -4682.694} C_VEL
LIN {X 0,Y 523.524,Z 265.801,A -85,B 0,C 180,E1 -4683.463,E2 -4683.463} C_VEL
LIN {X 0,Y 523.565,Z 261.143,A -85,B 0,C 180,E1 -4684.427,E2 -4684.427} C_VEL
LIN {X 0,Y 523.638,Z 256.235,A -85,B 0,C 180,E1 -4685.198,E2 -4685.198} C_VEL
LIN {X 0,Y 523.655,Z 250.01,A -85,B 0,C 180,E1 -4685.97,E2 -4685.97} C_VEL
LIN {X 0,Y 523.876,Z 241.554,A -85,B 0,C 180,E1 -4686.773,E2 -4686.773} C_VEL
LIN {X 0,Y 524.058,Z 232.486,A -85,B 0,C 180,E1 -4687.416,E2 -4687.416} C_VEL
LIN {X 0,Y 524.237,Z 223.169,A -85,B 0,C 180,E1 -4687.898,E2 -4687.898} C_VEL
LIN {X 0,Y 523.47,Z 214.736,A -85,B 0,C 180,E1 -4688.25,E2 -4688.25} C_VEL
LIN {X 0,Y 523.561,Z 205.844,A -85,B 0,C 180,E1 -4691.174,E2 -4691.174} C_VEL
LIN {X 0,Y 523.687,Z 196.22,A -85,B 0,C 180,E1 -4694.376,E2 -4694.376} C_VEL
LIN {X 0,Y 523.79,Z 187.871,A -85,B 0,C 180,E1 -4697.169,E2 -4697.169} C_VEL
LIN {X 0,Y 523.904,Z 180.718,A -85,B 0,C 180,E1 -4699.595,E2 -4699.595} C_VEL
LIN {X 0,Y 523.996,Z 172.947,A -85,B 0,C 180,E1 -4702.262,E2 -4702.262} C_VEL
LIN {X 0,Y 524.186,Z 163.936,A -85,B 0,C 180,E1 -4705.407,E2 -4705.407} C_VEL
LIN {X 0,Y 524.415,Z 156.674,A -85,B 0,C 180,E1 -4707.973,E2 -4707.973} C_VEL
LIN {X 0,Y 524.55,Z 150.646,A -85,B 0,C 180,E1 -4710.161,E2 -4710.161} C_VEL
LIN {X 0,Y 523.968,Z 147.223,A -85,B 0,C 180,E1 -4711.541,E2 -4711.541} C_VEL
LIN {X 0,Y 523.926,Z 147.226,A -85,B 0,C 180,E1 -4714.291,E2 -4714.291} C_VEL
LIN {X 0,Y 523.913,Z 147.228,A -85,B 0,C 180,E1 -4717.132,E2 -4717.132} C_VEL
LIN {X 0,Y 523.944,Z 147.223,A -85,B 0,C 180,E1 -4720.13,E2 -4720.13} C_VEL
LIN {X 0,Y 523.941,Z 147.225,A -85,B 0,C 180,E1 -4722.458,E2 -4722.458} C_VEL
LIN {X 0,Y 523.951,Z 147.222,A -85,B 0,C 180,E1 -4725.31,E2 -4725.31} C_VEL
LIN {X 0,Y 523.962,Z 147.22,A -85,B 0,C 180,E1 -4728.689,E2 -4728.689} C_VEL
LIN {X 0,Y 523.922,Z 147.227,A -85,B 0,C 180,E1 -4731.08,E2 -4731.08} C_VEL
LIN {X 0,Y 523.907,Z 147.228,A -85,B 0,C 180,E1 -4733.825,E2 -4733.825} C_VEL
LIN {X 0,Y 523.919,Z 147.228,A -85,B 0,C 180,E1 -4736.633,E2 -4736.633} C_VEL
LIN {X 0,Y 523.962,Z 147.226,A -85,B 0,C 180,E1 -4739.355,E2 -4739.355} C_VEL
LIN {X 0,Y 523.951,Z 147.296,A -85,B 0,C 180,E1 -4740.37,E2 -4740.37} C_VEL
LIN {X 0,Y 525.579,Z 155.094,A -85,B 0,C 180,E1 -4742.526,E2 -4742.526} C_VEL
LIN {X 0,Y 525.833,Z 159.293,A -85,B 0,C 180,E1 -4743.571,E2 -4743.571} C_VEL
LIN {X 0,Y 525.153,Z 171.412,A -85,B 0,C 180,E1 -4746.328,E2 -4746.328} C_VEL
LIN {X 0,Y 524.67,Z 184.824,A -85,B 0,C 180,E1 -4749.207,E2 -4749.207} C_VEL
LIN {X 0,Y 524.278,Z 200.856,A -85,B 0,C 180,E1 -4752.48,E2 -4752.48} C_VEL
LIN {X 0,Y 523.957,Z 216.845,A -85,B 0,C 180,E1 -4755.631,E2 -4755.631} C_VEL
LIN {X 0,Y 523.886,Z 220.755,A -85,B 0,C 180,E1 -4756.396,E2 -4756.396} C_VEL
LIN {X 0,Y 525.18,Z 231.861,A -85,B 0,C 180,E1 -4756.652,E2 -4756.652} C_VEL
LIN {X 0,Y 525.006,Z 244.595,A -85,B 0,C 180,E1 -4757.042,E2 -4757.042} C_VEL
LIN {X 0,Y 524.729,Z 256.968,A -85,B 0,C 180,E1 -4757.576,E2 -4757.576} C_VEL
LIN {X 0,Y 524.544,Z 269.119,A -85,B 0,C 180,E1 -4758.277,E2 -4758.277} C_VEL
LIN {X 0,Y 524.269,Z 280.086,A -85,B 0,C 180,E1 -4759.084,E2 -4759.084} C_VEL
LIN {X 0,Y 524.006,Z 289.704,A -85,B 0,C 180,E1 -4759.958,E2 -4759.958} C_VEL
LIN {X 0,Y 523.819,Z 298.467,A -85,B 0,C 180,E1 -4760.928,E2 -4760.928} C_VEL
LIN {X 0,Y 523.662,Z 306.939,A -85,B 0,C 180,E1 -4762.092,E2 -4762.092} C_VEL
LIN {X 0,Y 523.501,Z 313.782,A -85,B 0,C 180,E1 -4763.26,E2 -4763.26} C_VEL
LIN {X 0,Y 523.461,Z 319.983,A -85,B 0,C 180,E1 -4764.606,E2 -4764.606} C_VEL
LIN {X 0,Y 523.424,Z 324.02,A -85,B 0,C 180,E1 -4765.764,E2 -4765.764} C_VEL
LIN {X 0,Y 523.368,Z 326.995,A -85,B 0,C 180,E1 -4766.92,E2 -4766.92} C_VEL
LIN {X 0,Y 523.335,Z 328.414,A -85,B 0,C 180,E1 -4767.69,E2 -4767.69} C_VEL
LIN {X 0,Y 523.261,Z 330.041,A -85,B 0,C 180,E1 -4769.229,E2 -4769.229} C_VEL
LIN {X 0,Y 523.262,Z 330.266,A -85,B 0,C 180,E1 -4769.999,E2 -4769.999} C_VEL
LIN {X 0,Y 523.26,Z 330.051,A -85,B 0,C 180,E1 -4770.768,E2 -4770.768} C_VEL
LIN {X 0,Y 523.335,Z 328.442,A -85,B 0,C 180,E1 -4772.308,E2 -4772.308} C_VEL
LIN {X 0,Y 523.367,Z 327.033,A -85,B 0,C 180,E1 -4773.078,E2 -4773.078} C_VEL
LIN {X 0,Y 523.424,Z 324.072,A -85,B 0,C 180,E1 -4774.234,E2 -4774.234} C_VEL
LIN {X 0,Y 523.461,Z 320.052,A -85,B 0,C 180,E1 -4775.391,E2 -4775.391} C_VEL
LIN {X 0,Y 523.511,Z 314.772,A -85,B 0,C 180,E1 -4776.569,E2 -4776.569} C_VEL
LIN {X 0,Y 523.613,Z 308.316,A -85,B 0,C 180,E1 -4777.712,E2 -4777.712} C_VEL
LIN {X 0,Y 523.814,Z 300.161,A -85,B 0,C 180,E1 -4778.875,E2 -4778.875} C_VEL
LIN {X 0,Y 523.976,Z 291.819,A -85,B 0,C 180,E1 -4779.845,E2 -4779.845} C_VEL
LIN {X 0,Y 524.246,Z 281.576,A -85,B 0,C 180,E1 -4780.816,E2 -4780.816} C_VEL
LIN {X 0,Y 524.521,Z 270.06,A -85,B 0,C 180,E1 -4781.684,E2 -4781.684} C_VEL
LIN {X 0,Y 524.756,Z 258.506,A -85,B 0,C 180,E1 -4782.372,E2 -4782.372} C_VEL
LIN {X 0,Y 524.977,Z 246.653,A -85,B 0,C 180,E1 -4782.907,E2 -4782.907} C_VEL
LIN {X 0,Y 525.184,Z 232.974,A -85,B 0,C 180,E1 -4783.345,E2 -4783.345} C_VEL
LIN {X 0,Y 524.88,Z 228.114,A -85,B 0,C 180,E1 -4783.464,E2 -4783.464} C_VEL
LIN {X 0,Y 523.888,Z 220.889,A -85,B 0,C 180,E1 -4783.626,E2 -4783.626} C_VEL
LIN {X 0,Y 524.156,Z 206.034,A -85,B 0,C 180,E1 -4786.553,E2 -4786.553} C_VEL
LIN {X 0,Y 524.433,Z 192.795,A -85,B 0,C 180,E1 -4789.166,E2 -4789.166} C_VEL
LIN {X 0,Y 524.864,Z 179.029,A -85,B 0,C 180,E1 -4792.018,E2 -4792.018} C_VEL
LIN {X 0,Y 525.335,Z 165.258,A -85,B 0,C 180,E1 -4794.922,E2 -4794.922} C_VEL
LIN {X 0,Y 525.643,Z 157.173,A -85,B 0,C 180,E1 -4796.652,E2 -4796.652} C_VEL
LIN {X 0,Y 524.791,Z 151.481,A -85,B 0,C 180,E1 -4797.949,E2 -4797.949} C_VEL
LIN {X 0,Y 523.956,Z 147.223,A -85,B 0,C 180,E1 -4798.985,E2 -4798.985} C_VEL
LIN {X 0,Y 523.915,Z 147.224,A -85,B 0,C 180,E1 -4801.543,E2 -4801.543} C_VEL
LIN {X 0,Y 523.939,Z 147.224,A -85,B 0,C 180,E1 -4804.288,E2 -4804.288} C_VEL
LIN {X 0,Y 523.905,Z 147.226,A -85,B 0,C 180,E1 -4807.13,E2 -4807.13} C_VEL
LIN {X 0,Y 523.929,Z 147.22,A -85,B 0,C 180,E1 -4810.128,E2 -4810.128} C_VEL
LIN {X 0,Y 523.892,Z 147.225,A -85,B 0,C 180,E1 -4813.168,E2 -4813.168} C_VEL
LIN {X 0,Y 523.932,Z 147.224,A -85,B 0,C 180,E1 -4815.771,E2 -4815.771} C_VEL
LIN {X 0,Y 523.952,Z 147.221,A -85,B 0,C 180,E1 -4818.909,E2 -4818.909} C_VEL
LIN {X 0,Y 523.905,Z 147.224,A -85,B 0,C 180,E1 -4821.897,E2 -4821.897} C_VEL
LIN {X 0,Y 523.909,Z 147.222,A -85,B 0,C 180,E1 -4824.911,E2 -4824.911} C_VEL
LIN {X 0,Y 523.931,Z 147.226,A -85,B 0,C 180,E1 -4827.677,E2 -4827.677} C_VEL
LIN {X 0,Y 523.958,Z 147.22,A -85,B 0,C 180,E1 -4830.672,E2 -4830.672} C_VEL
LIN {X 0,Y 523.965,Z 147.217,A -85,B 0,C 180,E1 -4833.728,E2 -4833.728} C_VEL
LIN {X 0,Y 523.898,Z 147.226,A -85,B 0,C 180,E1 -4836.269,E2 -4836.269} C_VEL
LIN {X 0,Y 523.932,Z 147.22,A -85,B 0,C 180,E1 -4838.766,E2 -4838.766} C_VEL
LIN {X 0,Y 523.941,Z 147.223,A -85,B 0,C 180,E1 -4841.22,E2 -4841.22} C_VEL
LIN {X 0,Y 523.929,Z 147.221,A -85,B 0,C 180,E1 -4843.639,E2 -4843.639} C_VEL
LIN {X 0,Y 523.929,Z 147.225,A -85,B 0,C 180,E1 -4846.028,E2 -4846.028} C_VEL
LIN {X 0,Y 523.998,Z 147.211,A -85,B 0,C 180,E1 -4848.394,E2 -4848.394} C_VEL
LIN {X 0,Y 523.983,Z 147.215,A -85,B 0,C 180,E1 -4851.516,E2 -4851.516} C_VEL
LIN {X 0,Y 524.085,Z 147.206,A -85,B 0,C 180,E1 -4854.614,E2 -4854.614} C_VEL
LIN {X 0,Y 524.099,Z 147.204,A -85,B 0,C 180,E1 -4857.694,E2 -4857.694} C_VEL
LIN {X 0,Y 524.107,Z 147.2,A -85,B 0,C 180,E1 -4860.768,E2 -4860.768} C_VEL
LIN {X 0,Y 524.051,Z 147.208,A -85,B 0,C 180,E1 -4863.075,E2 -4863.075} C_VEL
LIN {X 0,Y 524.03,Z 147.212,A -85,B 0,C 180,E1 -4866.159,E2 -4866.159} C_VEL
LIN {X 0,Y 523.992,Z 147.216,A -85,B 0,C 180,E1 -4869.262,E2 -4869.262} C_VEL
LIN {X 0,Y 524.009,Z 147.211,A -85,B 0,C 180,E1 -4871.752,E2 -4871.752} C_VEL
LIN {X 0,Y 523.978,Z 147.214,A -85,B 0,C 180,E1 -4875.053,E2 -4875.053} C_VEL
LIN {X 0,Y 523.95,Z 147.223,A -85,B 0,C 180,E1 -4877.969,E2 -4877.969} C_VEL
LIN {X 0,Y 523.959,Z 147.217,A -85,B 0,C 180,E1 -4880.411,E2 -4880.411} C_VEL
LIN {X 0,Y 523.931,Z 147.225,A -85,B 0,C 180,E1 -4882.893,E2 -4882.893} C_VEL
LIN {X 0,Y 523.922,Z 147.221,A -85,B 0,C 180,E1 -4885.42,E2 -4885.42} C_VEL
LIN {X 0,Y 523.903,Z 147.229,A -85,B 0,C 180,E1 -4888.003,E2 -4888.003} C_VEL
LIN {X 0,Y 523.94,Z 147.22,A -85,B 0,C 180,E1 -4890.857,E2 -4890.857} C_VEL
LIN {X 0,Y 523.951,Z 147.218,A -85,B 0,C 180,E1 -4893.736,E2 -4893.736} C_VEL
LIN {X 0,Y 523.911,Z 147.227,A -85,B 0,C 180,E1 -4896.405,E2 -4896.405} C_VEL
LIN {X 0,Y 523.907,Z 147.223,A -85,B 0,C 180,E1 -4899.086,E2 -4899.086} C_VEL
LIN {X 0,Y 523.941,Z 147.219,A -85,B 0,C 180,E1 -4902.12,E2 -4902.12} C_VEL
LIN {X 0,Y 523.947,Z 147.22,A -85,B 0,C 180,E1 -4905.31,E2 -4905.31} C_VEL
LIN {X 0,Y 523.914,Z 147.224,A -85,B 0,C 180,E1 -4906.932,E2 -4906.932} C_VEL
LIN {X 0,Y 523.247,Z 147.307,A -85,B 0,C 180,E1 -4907.574,E2 -4907.574} C_VEL
LIN {X 0,Y 520.403,Z 147.661,A -85,B 0,C 180,E1 -4908.616,E2 -4908.616} C_VEL
LIN {X 0,Y 517.996,Z 147.963,A -85,B 0,C 180,E1 -4909.454,E2 -4909.454} C_VEL
LIN {X 0,Y 516.958,Z 148.091,A -85,B 0,C 180,E1 -4910.102,E2 -4910.102} C_VEL
LIN {X 0,Y 516.872,Z 148.1,A -85,B 0,C 180,E1 -4910.322,E2 -4910.322} C_VEL
LIN {X 0,Y 516.845,Z 148.107,A -85,B 0,C 180,E1 -4913.348,E2 -4913.348} C_VEL
LIN {X 0,Y 516.901,Z 148.097,A -85,B 0,C 180,E1 -4916.122,E2 -4916.122} C_VEL
LIN {X 0,Y 516.889,Z 148.098,A -85,B 0,C 180,E1 -4918.936,E2 -4918.936} C_VEL
LIN {X 0,Y 516.917,Z 148.098,A -85,B 0,C 180,E1 -4921.586,E2 -4921.586} C_VEL
LIN {X 0,Y 516.886,Z 148.097,A -85,B 0,C 180,E1 -4924.21,E2 -4924.21} C_VEL
LIN {X 0,Y 516.852,Z 148.106,A -85,B 0,C 180,E1 -4926.777,E2 -4926.777} C_VEL
LIN {X 0,Y 516.937,Z 148.095,A -85,B 0,C 180,E1 -4929.733,E2 -4929.733} C_VEL
LIN {X 0,Y 516.928,Z 148.093,A -85,B 0,C 180,E1 -4932.598,E2 -4932.598} C_VEL
LIN {X 0,Y 516.938,Z 148.096,A -85,B 0,C 180,E1 -4935.031,E2 -4935.031} C_VEL
LIN {X 0,Y 516.966,Z 148.092,A -85,B 0,C 180,E1 -4938.235,E2 -4938.235} C_VEL
LIN {X 0,Y 516.964,Z 148.09,A -85,B 0,C 180,E1 -4941.401,E2 -4941.401} C_VEL
LIN {X 0,Y 517.012,Z 148.085,A -85,B 0,C 180,E1 -4943.758,E2 -4943.758} C_VEL
LIN {X 0,Y 517.085,Z 148.073,A -85,B 0,C 180,E1 -4947.664,E2 -4947.664} C_VEL
LIN {X 0,Y 517.068,Z 148.08,A -85,B 0,C 180,E1 -4950.001,E2 -4950.001} C_VEL
LIN {X 0,Y 517.081,Z 148.074,A -85,B 0,C 180,E1 -4952.338,E2 -4952.338} C_VEL
LIN {X 0,Y 517.014,Z 148.083,A -85,B 0,C 180,E1 -4956.244,E2 -4956.244} C_VEL
LIN {X 0,Y 516.947,Z 148.09,A -85,B 0,C 180,E1 -4959.39,E2 -4959.39} C_VEL
LIN {X 0,Y 516.956,Z 148.095,A -85,B 0,C 180,E1 -4961.808,E2 -4961.808} C_VEL
LIN {X 0,Y 516.939,Z 148.095,A -85,B 0,C 180,E1 -4965.143,E2 -4965.143} C_VEL
LIN {X 0,Y 516.921,Z 148.096,A -85,B 0,C 180,E1 -4968.223,E2 -4968.223} C_VEL
LIN {X 0,Y 516.917,Z 148.096,A -85,B 0,C 180,E1 -4970.702,E2 -4970.702} C_VEL
LIN {X 0,Y 516.888,Z 148.098,A -85,B 0,C 180,E1 -4974.074,E2 -4974.074} C_VEL
LIN {X 0,Y 516.843,Z 148.104,A -85,B 0,C 180,E1 -4976.663,E2 -4976.663} C_VEL
LIN {X 0,Y 516.891,Z 148.097,A -85,B 0,C 180,E1 -4979.519,E2 -4979.519} C_VEL
LIN {X 0,Y 516.899,Z 148.097,A -85,B 0,C 180,E1 -4982.544,E2 -4982.544} C_VEL
LIN {X 0,Y 516.868,Z 148.105,A -85,B 0,C 180,E1 -4985.33,E2 -4985.33} C_VEL
LIN {X 0,Y 516.858,Z 148.1,A -85,B 0,C 180,E1 -4987.94,E2 -4987.94} C_VEL
LIN {X 0,Y 516.858,Z 148.103,A -85,B 0,C 180,E1 -4990.745,E2 -4990.745} C_VEL
LIN {X 0,Y 516.862,Z 148.101,A -85,B 0,C 180,E1 -4992.835,E2 -4992.835} C_VEL
LIN {X 0,Y 516.9,Z 148.098,A -85,B 0,C 180,E1 -4995.007,E2 -4995.007} C_VEL
LIN {X 0,Y 516.918,Z 148.096,A -85,B 0,C 180,E1 -4998.399,E2 -4998.399} C_VEL
LIN {X 0,Y 516.876,Z 148.098,A -85,B 0,C 180,E1 -5001.284,E2 -5001.284} C_VEL
LIN {X 0,Y 516.867,Z 148.1,A -85,B 0,C 180,E1 -5004.671,E2 -5004.671} C_VEL
LIN {X 0,Y 516.899,Z 148.101,A -85,B 0,C 180,E1 -5007.457,E2 -5007.457} C_VEL
LIN {X 0,Y 516.982,Z 148.193,A -85,B 0,C 180,E1 -5008.84,E2 -5008.84} C_VEL
LIN {X 0,Y 517.393,Z 152.35,A -85,B 0,C 180,E1 -5010.384,E2 -5010.384} C_VEL
LIN {X 0,Y 517.197,Z 161.739,A -85,B 0,C 180,E1 -5013.748,E2 -5013.748} C_VEL
LIN {X 0,Y 516.976,Z 170.35,A -85,B 0,C 180,E1 -5016.782,E2 -5016.782} C_VEL
LIN {X 0,Y 516.835,Z 178.964,A -85,B 0,C 180,E1 -5019.765,E2 -5019.765} C_VEL
LIN {X 0,Y 516.709,Z 188.468,A -85,B 0,C 180,E1 -5022.996,E2 -5022.996} C_VEL
LIN {X 0,Y 516.573,Z 196.772,A -85,B 0,C 180,E1 -5025.825,E2 -5025.825} C_VEL
LIN {X 0,Y 516.488,Z 204.518,A -85,B 0,C 180,E1 -5028.445,E2 -5028.445} C_VEL
LIN {X 0,Y 516.385,Z 214.062,A -85,B 0,C 180,E1 -5031.587,E2 -5031.587} C_VEL
LIN {X 0,Y 516.374,Z 214.588,A -85,B 0,C 180,E1 -5031.759,E2 -5031.759} C_VEL
LIN {X 0,Y 517.169,Z 224.042,A -85,B 0,C 180,E1 -5032.141,E2 -5032.141} C_VEL
